IF NOT _DispatchValid() THEN
	RETURN;
ELSE
	_BuildCommandStringNoArgs();
	
	IF iBufferSend <> 0 AND __QUERYINTERFACE(iBufferSend, testIBufferSend) THEN
		iBufferSend.AddObject(RefObject := ZaberCommand);
	END_IF
END_IF
END_METHOD

METHOD set_user_vdata_3
IF ZaberStatus.ComponentStatus.iLastCommand <> 0 THEN
	ZaberStatus.ComponentStatus.iLastCommand.P_CommandStatus.LastCommandMessage := Base.F_GetLastWordInString(__POUNAME());
END_IF

IF NOT _DispatchValid() THEN
	RETURN;
ELSE
	_BuildCommandStringNoArgs();
	
	IF iBufferSend <> 0 AND __QUERYINTERFACE(iBufferSend, testIBufferSend) THEN
		iBufferSend.AddObject(RefObject := ZaberCommand);
	END_IF
END_IF
END_METHOD

METHOD set_vel
IF ZaberStatus.ComponentStatus.iLastCommand <> 0 THEN
	ZaberStatus.ComponentStatus.iLastCommand.P_CommandStatus.LastCommandMessage := Base.F_GetLastWordInString(__POUNAME());
END_IF

IF NOT _DispatchValid() THEN
	RETURN;
ELSE
	_BuildCommandStringNoArgs();
	
	IF iBufferSend <> 0 AND __QUERYINTERFACE(iBufferSend, testIBufferSend) THEN
		iBufferSend.AddObject(RefObject := ZaberCommand);
	END_IF
END_IF
END_METHOD

METHOD set_version
IF ZaberStatus.ComponentStatus.iLastCommand <> 0 THEN
	ZaberStatus.ComponentStatus.iLastCommand.P_CommandStatus.LastCommandMessage := Base.F_GetLastWordInString(__POUNAME());
END_IF

IF NOT _DispatchValid() THEN
	RETURN;
ELSE
	_BuildCommandStringNoArgs();
	
	IF iBufferSend <> 0 AND __QUERYINTERFACE(iBufferSend, testIBufferSend) THEN
		iBufferSend.AddObject(RefObject := ZaberCommand);
	END_IF
END_IF
END_METHOD

METHOD set_version_build
IF ZaberStatus.ComponentStatus.iLastCommand <> 0 THEN
	ZaberStatus.ComponentStatus.iLastCommand.P_CommandStatus.LastCommandMessage := Base.F_GetLastWordInString(__POUNAME());
END_IF

IF NOT _DispatchValid() THEN
	RETURN;
ELSE
	_BuildCommandStringNoArgs();
	
	IF iBufferSend <> 0 AND __QUERYINTERFACE(iBufferSend, testIBufferSend) THEN
		iBufferSend.AddObject(RefObject := ZaberCommand);
	END_IF
END_IF
END_METHOD

METHOD storage_append
IF ZaberStatus.ComponentStatus.iLastCommand <> 0 THEN
	ZaberStatus.ComponentStatus.iLastCommand.P_CommandStatus.LastCommandMessage := Base.F_GetLastWordInString(__POUNAME());
END_IF

IF NOT _DispatchValid() THEN
	RETURN;
ELSE
	_BuildCommandStringNoArgs();
	
	IF iBufferSend <> 0 AND __QUERYINTERFACE(iBufferSend, testIBufferSend) THEN
		iBufferSend.AddObject(RefObject := ZaberCommand);
	END_IF
END_IF
END_METHOD

METHOD storage_exists
IF ZaberStatus.ComponentStatus.iLastCommand <> 0 THEN
	ZaberStatus.ComponentStatus.iLastCommand.P_CommandStatus.LastCommandMessage := Base.F_GetLastWordInString(__POUNAME());
END_IF

IF NOT _DispatchValid() THEN
	RETURN;
ELSE
	_BuildCommandStringNoArgs();
	
	IF iBufferSend <> 0 AND __QUERYINTERFACE(iBufferSend, testIBufferSend) THEN
		iBufferSend.AddObject(RefObject := ZaberCommand);
	END_IF
END_IF
END_METHOD

METHOD storage_get
IF ZaberStatus.ComponentStatus.iLastCommand <> 0 THEN
	ZaberStatus.ComponentStatus.iLastCommand.P_CommandStatus.LastCommandMessage := Base.F_GetLastWordInString(__POUNAME());
END_IF

IF NOT _DispatchValid() THEN
	RETURN;
ELSE
	_BuildCommandStringNoArgs();
	
	IF iBufferSend <> 0 AND __QUERYINTERFACE(iBufferSend, testIBufferSend) THEN
		iBufferSend.AddObject(RefObject := ZaberCommand);
	END_IF
END_IF
END_METHOD

METHOD storage_set
IF ZaberStatus.ComponentStatus.iLastCommand <> 0 THEN
	ZaberStatus.ComponentStatus.iLastCommand.P_CommandStatus.LastCommandMessage := Base.F_GetLastWordInString(__POUNAME());
END_IF

IF NOT _DispatchValid() THEN
	RETURN;
ELSE
	_BuildCommandStringNoArgs();
	
	IF iBufferSend <> 0 AND __QUERYINTERFACE(iBufferSend, testIBufferSend) THEN
		iBufferSend.AddObject(RefObject := ZaberCommand);
	END_IF
END_IF
END_METHOD

//stream <number> [on <axis1> <axis2>] arc abs|rel cw|ccw <centrex> <centrey> <endx> <endy> [join maxspeed <speed>]; Creates an arc path segment
METHOD stream_arc
VAR_INPUT
	StreamIndex : UDINT; //<number> The number OF the stream TO ADD the ACTION TO.  Must be in the range 1 TO stream.numstreams
	Axis1 : UINT; //<axis1> The first stream axis on which TO execute the arc segment (optional).  The first stream axis is labelled "a", the second "b", AND so on
	Axis2 : UINT; //<axis2> The second stream axis on which to execute the arc segment (optional). The first stream axis is labelled "a", the second "b", and so on
	MoveType : E_MoveType; //abs Indicates that position parameters are absolute positions; rel Indicates that position parameters are relative to the end point of the previous path segment
	Direction : E_MoveDirection; //cw Indicates that the arc should be in the clockwise direction; //ccw Indicates that the arc should be in the counter-clockwise direction
	CenterX : DINT; //<centrex> The x-axis position of the arc�s centre; Must be the range -2,147,483,648 to 2,147,483,647
	CenterY : DINT; //<centrey> The y-axis position of the arc�s centre; Must be the range -2,147,483,648 to 2,147,483,647
	EndX : DINT; //<endx> The x-axis position of the end of the arc; Must be in the range limit.min to limit.max for that axis
	EndY : DINT; //<endy> The y-axis position of the end of the arc; Must be in the range limit.min to limit.max for that axis
	Speed : UDINT; //<speed> The speed LIMIT FOR the transition between the previous segment AND THIS one (optional); Must be in the range 0 TO resolution � 16,384 FOR stepper motor products; Must be in the range 0 TO 4,294,967,295 FOR linear motor OR voice coil products
END_VAR
IF ZaberStatus.ComponentStatus.iLastCommand <> 0 THEN
	ZaberStatus.ComponentStatus.iLastCommand.P_CommandStatus.LastCommandMessage := Base.F_GetLastWordInString(__POUNAME());
END_IF

IF NOT _DispatchValid() THEN
	RETURN;
ELSE
	_BuildCommandStringNoArgs();
	
	IF iBufferSend <> 0 AND __QUERYINTERFACE(iBufferSend, testIBufferSend) THEN
		iBufferSend.AddObject(RefObject := ZaberCommand);
	END_IF
END_IF
END_METHOD

METHOD stream_buffer_erase
IF ZaberStatus.ComponentStatus.iLastCommand <> 0 THEN
	ZaberStatus.ComponentStatus.iLastCommand.P_CommandStatus.LastCommandMessage := Base.F_GetLastWordInString(__POUNAME());
END_IF

IF NOT _DispatchValid() THEN
	RETURN;
ELSE
	_BuildCommandStringNoArgs();
	
	IF iBufferSend <> 0 AND __QUERYINTERFACE(iBufferSend, testIBufferSend) THEN
		iBufferSend.AddObject(RefObject := ZaberCommand);
	END_IF
END_IF
END_METHOD

METHOD stream_buffer_print
IF ZaberStatus.ComponentStatus.iLastCommand <> 0 THEN
	ZaberStatus.ComponentStatus.iLastCommand.P_CommandStatus.LastCommandMessage := Base.F_GetLastWordInString(__POUNAME());
END_IF

IF NOT _DispatchValid() THEN
	RETURN;
ELSE
	_BuildCommandStringNoArgs();
	
	IF iBufferSend <> 0 AND __QUERYINTERFACE(iBufferSend, testIBufferSend) THEN
		iBufferSend.AddObject(RefObject := ZaberCommand);
	END_IF
END_IF
END_METHOD

METHOD stream_call
IF ZaberStatus.ComponentStatus.iLastCommand <> 0 THEN
	ZaberStatus.ComponentStatus.iLastCommand.P_CommandStatus.LastCommandMessage := Base.F_GetLastWordInString(__POUNAME());
END_IF

IF NOT _DispatchValid() THEN
	RETURN;
ELSE
	_BuildCommandStringNoArgs();
	
	IF iBufferSend <> 0 AND __QUERYINTERFACE(iBufferSend, testIBufferSend) THEN
		iBufferSend.AddObject(RefObject := ZaberCommand);
	END_IF
END_IF
END_METHOD

METHOD stream_circle
IF ZaberStatus.ComponentStatus.iLastCommand <> 0 THEN
	ZaberStatus.ComponentStatus.iLastCommand.P_CommandStatus.LastCommandMessage := Base.F_GetLastWordInString(__POUNAME());
END_IF

IF NOT _DispatchValid() THEN
	RETURN;
ELSE
	_BuildCommandStringNoArgs();
	
	IF iBufferSend <> 0 AND __QUERYINTERFACE(iBufferSend, testIBufferSend) THEN
		iBufferSend.AddObject(RefObject := ZaberCommand);
	END_IF
END_IF
END_METHOD

METHOD stream_fifo
IF ZaberStatus.ComponentStatus.iLastCommand <> 0 THEN
	ZaberStatus.ComponentStatus.iLastCommand.P_CommandStatus.LastCommandMessage := Base.F_GetLastWordInString(__POUNAME());
END_IF

IF NOT _DispatchValid() THEN
	RETURN;
ELSE
	_BuildCommandStringNoArgs();
	
	IF iBufferSend <> 0 AND __QUERYINTERFACE(iBufferSend, testIBufferSend) THEN
		iBufferSend.AddObject(RefObject := ZaberCommand);
	END_IF
END_IF
END_METHOD

METHOD stream_helix
IF ZaberStatus.ComponentStatus.iLastCommand <> 0 THEN
	ZaberStatus.ComponentStatus.iLastCommand.P_CommandStatus.LastCommandMessage := Base.F_GetLastWordInString(__POUNAME());
END_IF

IF NOT _DispatchValid() THEN
	RETURN;
ELSE
	_BuildCommandStringNoArgs();
	
	IF iBufferSend <> 0 AND __QUERYINTERFACE(iBufferSend, testIBufferSend) THEN
		iBufferSend.AddObject(RefObject := ZaberCommand);
	END_IF
END_IF
END_METHOD

METHOD stream_hold_onloff
IF ZaberStatus.ComponentStatus.iLastCommand <> 0 THEN
	ZaberStatus.ComponentStatus.iLastCommand.P_CommandStatus.LastCommandMessage := Base.F_GetLastWordInString(__POUNAME());
END_IF

IF NOT _DispatchValid() THEN
	RETURN;
ELSE
	_BuildCommandStringNoArgs();
	
	IF iBufferSend <> 0 AND __QUERYINTERFACE(iBufferSend, testIBufferSend) THEN
		iBufferSend.AddObject(RefObject := ZaberCommand);
	END_IF
END_IF
END_METHOD

METHOD stream_info
IF ZaberStatus.ComponentStatus.iLastCommand <> 0 THEN
	ZaberStatus.ComponentStatus.iLastCommand.P_CommandStatus.LastCommandMessage := Base.F_GetLastWordInString(__POUNAME());
END_IF

IF NOT _DispatchValid() THEN
	RETURN;
ELSE
	_BuildCommandStringNoArgs();
	
	IF iBufferSend <> 0 AND __QUERYINTERFACE(iBufferSend, testIBufferSend) THEN
		iBufferSend.AddObject(RefObject := ZaberCommand);
	END_IF
END_IF
END_METHOD

METHOD stream_io_cancel_schedule
IF ZaberStatus.ComponentStatus.iLastCommand <> 0 THEN
	ZaberStatus.ComponentStatus.iLastCommand.P_CommandStatus.LastCommandMessage := Base.F_GetLastWordInString(__POUNAME());
END_IF

IF NOT _DispatchValid() THEN
	RETURN;
ELSE
	_BuildCommandStringNoArgs();
	
	IF iBufferSend <> 0 AND __QUERYINTERFACE(iBufferSend, testIBufferSend) THEN
		iBufferSend.AddObject(RefObject := ZaberCommand);
	END_IF
END_IF
END_METHOD

METHOD stream_io_set_ao
IF ZaberStatus.ComponentStatus.iLastCommand <> 0 THEN
	ZaberStatus.ComponentStatus.iLastCommand.P_CommandStatus.LastCommandMessage := Base.F_GetLastWordInString(__POUNAME());
END_IF

IF NOT _DispatchValid() THEN
	RETURN;
ELSE
	_BuildCommandStringNoArgs();
	
	IF iBufferSend <> 0 AND __QUERYINTERFACE(iBufferSend, testIBufferSend) THEN
		iBufferSend.AddObject(RefObject := ZaberCommand);
	END_IF
END_IF
END_METHOD

METHOD stream_io_set_ao_schedule
IF ZaberStatus.ComponentStatus.iLastCommand <> 0 THEN
	ZaberStatus.ComponentStatus.iLastCommand.P_CommandStatus.LastCommandMessage := Base.F_GetLastWordInString(__POUNAME());
END_IF

IF NOT _DispatchValid() THEN
	RETURN;
ELSE
	_BuildCommandStringNoArgs();
	
	IF iBufferSend <> 0 AND __QUERYINTERFACE(iBufferSend, testIBufferSend) THEN
		iBufferSend.AddObject(RefObject := ZaberCommand);
	END_IF
END_IF
END_METHOD

METHOD stream_io_set_do
IF ZaberStatus.ComponentStatus.iLastCommand <> 0 THEN
	ZaberStatus.ComponentStatus.iLastCommand.P_CommandStatus.LastCommandMessage := Base.F_GetLastWordInString(__POUNAME());
END_IF

IF NOT _DispatchValid() THEN
	RETURN;
ELSE
	_BuildCommandStringNoArgs();
	
	IF iBufferSend <> 0 AND __QUERYINTERFACE(iBufferSend, testIBufferSend) THEN
		iBufferSend.AddObject(RefObject := ZaberCommand);
	END_IF
END_IF
END_METHOD

METHOD stream_io_set_do_schedule
IF ZaberStatus.ComponentStatus.iLastCommand <> 0 THEN
	ZaberStatus.ComponentStatus.iLastCommand.P_CommandStatus.LastCommandMessage := Base.F_GetLastWordInString(__POUNAME());
END_IF

IF NOT _DispatchValid() THEN
	RETURN;
ELSE
	_BuildCommandStringNoArgs();
	
	IF iBufferSend <> 0 AND __QUERYINTERFACE(iBufferSend, testIBufferSend) THEN
		iBufferSend.AddObject(RefObject := ZaberCommand);
	END_IF
END_IF
END_METHOD

METHOD stream_line
IF ZaberStatus.ComponentStatus.iLastCommand <> 0 THEN
	ZaberStatus.ComponentStatus.iLastCommand.P_CommandStatus.LastCommandMessage := Base.F_GetLastWordInString(__POUNAME());
END_IF

IF NOT _DispatchValid() THEN
	RETURN;
ELSE
	_BuildCommandStringNoArgs();
	
	IF iBufferSend <> 0 AND __QUERYINTERFACE(iBufferSend, testIBufferSend) THEN
		iBufferSend.AddObject(RefObject := ZaberCommand);
	END_IF
END_IF
END_METHOD

METHOD stream_set
IF ZaberStatus.ComponentStatus.iLastCommand <> 0 THEN
	ZaberStatus.ComponentStatus.iLastCommand.P_CommandStatus.LastCommandMessage := Base.F_GetLastWordInString(__POUNAME());
END_IF

IF NOT _DispatchValid() THEN
	RETURN;
ELSE
	_BuildCommandStringNoArgs();
	
	IF iBufferSend <> 0 AND __QUERYINTERFACE(iBufferSend, testIBufferSend) THEN
		iBufferSend.AddObject(RefObject := ZaberCommand);
	END_IF
END_IF
END_METHOD

METHOD stream_setup_disable
IF ZaberStatus.ComponentStatus.iLastCommand <> 0 THEN
	ZaberStatus.ComponentStatus.iLastCommand.P_CommandStatus.LastCommandMessage := Base.F_GetLastWordInString(__POUNAME());
END_IF

IF NOT _DispatchValid() THEN
	RETURN;
ELSE
	_BuildCommandStringNoArgs();
	
	IF iBufferSend <> 0 AND __QUERYINTERFACE(iBufferSend, testIBufferSend) THEN
		iBufferSend.AddObject(RefObject := ZaberCommand);
	END_IF
END_IF
END_METHOD

METHOD stream_setup_live
VAR_INPUT
	StreamNumber : UDINT;
	AxisNumber : UDINT;
END_VAR
IF ZaberStatus.ComponentStatus.iLastCommand <> 0 THEN
	ZaberStatus.ComponentStatus.iLastCommand.P_CommandStatus.LastCommandMessage := Base.F_GetLastWordInString(__POUNAME());
END_IF

IF NOT _DispatchValid() THEN
	RETURN;
ELSE
	_ClearTempString();
	ZaberCommand.stringval := Tc2_Standard.CONCAT(STR1 := ZaberConfiguration.sControllerRef, STR2 := ' ');
	ZaberCommand.stringval := Tc2_Standard.CONCAT(STR1 := ZaberCommand.stringval, STR2 := UINT_TO_STRING(ZaberConfiguration.AxisRef));
	ZaberCommand.stringval := Tc2_Standard.CONCAT(STR1 := ZaberCommand.stringval, STR2 := ' ');
	ZaberCommand.stringval := Tc2_Standard.CONCAT(STR1 := ZaberCommand.stringval, STR2 := Base.F_GetFirstWordInString(SUPER^._iCommandConfiguration[ZaberStatus.ZaberMethodDispatch].P_CommandConfiguration.CommandDescription));
	ZaberCommand.stringval := Tc2_Standard.CONCAT(STR1 := ZaberCommand.stringval, STR2 := ' ');
	ZaberCommand.stringval := Tc2_Standard.CONCAT(STR1 := ZaberCommand.stringval, STR2 := UDINT_TO_STRING(StreamNumber));
	ZaberCommand.stringval := Tc2_Standard.CONCAT(STR1 := ZaberCommand.stringval, STR2 := ' ');
	ZaberCommand.stringval := Tc2_Standard.CONCAT(STR1 := ZaberCommand.stringval, STR2 := F_GetAllButFirstWord(SUPER^._iCommandConfiguration[ZaberStatus.ZaberMethodDispatch].P_CommandConfiguration.CommandDescription));
	ZaberCommand.stringval := Tc2_Standard.CONCAT(STR1 := ZaberCommand.stringval, STR2 := ' ');
	ZaberCommand.stringval := Tc2_Standard.CONCAT(STR1 := ZaberCommand.stringval, STR2 := UDINT_TO_STRING(AxisNumber));

	IF iBufferSend <> 0 AND __QUERYINTERFACE(iBufferSend, testIBufferSend) THEN
		iBufferSend.AddObject(RefObject := ZaberCommand);
	END_IF
END_IF
END_METHOD

METHOD stream_setup_store
VAR_INPUT
	StreamNumber	: UDINT; //The number OF the stream TO enable; Must be in the range 1 TO stream.numstreams
	BufferNumber	: UDINT; //The number OF the buffer TO write TO; Must be in the range 1 to stream.numbufs
	AxisNumber		: UINT; //The number OF axes in the path ; Must be in the range 1 TO system.axiscount
END_VAR
IF ZaberStatus.ComponentStatus.iLastCommand <> 0 THEN
	ZaberStatus.ComponentStatus.iLastCommand.P_CommandStatus.LastCommandMessage := Base.F_GetLastWordInString(__POUNAME());
END_IF

IF NOT _DispatchValid() THEN
	RETURN;
ELSE
	_ClearTempString();
	ZaberCommand.stringval := Tc2_Standard.CONCAT(STR1 := ZaberConfiguration.sControllerRef, STR2 := ' ');
	ZaberCommand.stringval := Tc2_Standard.CONCAT(STR1 := ZaberCommand.stringval, STR2 := UINT_TO_STRING(ZaberConfiguration.AxisRef));
	ZaberCommand.stringval := Tc2_Standard.CONCAT(STR1 := ZaberCommand.stringval, STR2 := ' ');
	ZaberCommand.stringval := Tc2_Standard.CONCAT(STR1 := ZaberCommand.stringval, STR2 := Base.F_GetFirstWordInString(SUPER^._iCommandConfiguration[ZaberStatus.ZaberMethodDispatch].P_CommandConfiguration.CommandDescription));
	ZaberCommand.stringval := Tc2_Standard.CONCAT(STR1 := ZaberCommand.stringval, STR2 := ' ');
	ZaberCommand.stringval := Tc2_Standard.CONCAT(STR1 := ZaberCommand.stringval, STR2 := UDINT_TO_STRING(StreamNumber));
	ZaberCommand.stringval := Tc2_Standard.CONCAT(STR1 := ZaberCommand.stringval, STR2 := ' ');
	ZaberCommand.stringval := Tc2_Standard.CONCAT(STR1 := ZaberCommand.stringval, STR2 := F_GetAllButFirstWord(SUPER^._iCommandConfiguration[ZaberStatus.ZaberMethodDispatch].P_CommandConfiguration.CommandDescription));
	ZaberCommand.stringval := Tc2_Standard.CONCAT(STR1 := ZaberCommand.stringval, STR2 := ' ');
	ZaberCommand.stringval := Tc2_Standard.CONCAT(STR1 := ZaberCommand.stringval, STR2 := UDINT_TO_STRING(BufferNumber));
	ZaberCommand.stringval := Tc2_Standard.CONCAT(STR1 := ZaberCommand.stringval, STR2 := ' ');
	ZaberCommand.stringval := Tc2_Standard.CONCAT(STR1 := ZaberCommand.stringval, STR2 := UINT_TO_STRING(AxisNumber));
	
	IF iBufferSend <> 0 AND __QUERYINTERFACE(iBufferSend, testIBufferSend) THEN
		iBufferSend.AddObject(RefObject := ZaberCommand);
	END_IF
END_IF
END_METHOD

METHOD stream_wait
IF ZaberStatus.ComponentStatus.iLastCommand <> 0 THEN
	ZaberStatus.ComponentStatus.iLastCommand.P_CommandStatus.LastCommandMessage := Base.F_GetLastWordInString(__POUNAME());
END_IF

IF NOT _DispatchValid() THEN
	RETURN;
ELSE
	_BuildCommandStringNoArgs();
	
	IF iBufferSend <> 0 AND __QUERYINTERFACE(iBufferSend, testIBufferSend) THEN
		iBufferSend.AddObject(RefObject := ZaberCommand);
	END_IF
END_IF
END_METHOD

METHOD stream_wait_io
IF ZaberStatus.ComponentStatus.iLastCommand <> 0 THEN
	ZaberStatus.ComponentStatus.iLastCommand.P_CommandStatus.LastCommandMessage := Base.F_GetLastWordInString(__POUNAME());
END_IF

IF NOT _DispatchValid() THEN
	RETURN;
ELSE
	_BuildCommandStringNoArgs();
	
	IF iBufferSend <> 0 AND __QUERYINTERFACE(iBufferSend, testIBufferSend) THEN
		iBufferSend.AddObject(RefObject := ZaberCommand);
	END_IF
END_IF
END_METHOD

METHOD tools_storepos
IF ZaberStatus.ComponentStatus.iLastCommand <> 0 THEN
	ZaberStatus.ComponentStatus.iLastCommand.P_CommandStatus.LastCommandMessage := Base.F_GetLastWordInString(__POUNAME());
END_IF

IF NOT _DispatchValid() THEN
	RETURN;
ELSE
	_BuildCommandStringNoArgs();
	
	IF iBufferSend <> 0 AND __QUERYINTERFACE(iBufferSend, testIBufferSend) THEN
		iBufferSend.AddObject(RefObject := ZaberCommand);
	END_IF
END_IF
END_METHOD

METHOD trigger_action_command
IF ZaberStatus.ComponentStatus.iLastCommand <> 0 THEN
	ZaberStatus.ComponentStatus.iLastCommand.P_CommandStatus.LastCommandMessage := Base.F_GetLastWordInString(__POUNAME());
END_IF

IF NOT _DispatchValid() THEN
	RETURN;
ELSE
	_BuildCommandStringNoArgs();
	
	IF iBufferSend <> 0 AND __QUERYINTERFACE(iBufferSend, testIBufferSend) THEN
		iBufferSend.AddObject(RefObject := ZaberCommand);
	END_IF
END_IF
END_METHOD

METHOD trigger_action_none
IF ZaberStatus.ComponentStatus.iLastCommand <> 0 THEN
	ZaberStatus.ComponentStatus.iLastCommand.P_CommandStatus.LastCommandMessage := Base.F_GetLastWordInString(__POUNAME());
END_IF

IF NOT _DispatchValid() THEN
	RETURN;
ELSE
	_BuildCommandStringNoArgs();
	
	IF iBufferSend <> 0 AND __QUERYINTERFACE(iBufferSend, testIBufferSend) THEN
		iBufferSend.AddObject(RefObject := ZaberCommand);
	END_IF
END_IF
END_METHOD

METHOD trigger_action_setting
IF ZaberStatus.ComponentStatus.iLastCommand <> 0 THEN
	ZaberStatus.ComponentStatus.iLastCommand.P_CommandStatus.LastCommandMessage := Base.F_GetLastWordInString(__POUNAME());
END_IF

IF NOT _DispatchValid() THEN
	RETURN;
ELSE
	_BuildCommandStringNoArgs();
	
	IF iBufferSend <> 0 AND __QUERYINTERFACE(iBufferSend, testIBufferSend) THEN
		iBufferSend.AddObject(RefObject := ZaberCommand);
	END_IF
END_IF
END_METHOD

METHOD trigger_disable
IF ZaberStatus.ComponentStatus.iLastCommand <> 0 THEN
	ZaberStatus.ComponentStatus.iLastCommand.P_CommandStatus.LastCommandMessage := Base.F_GetLastWordInString(__POUNAME());
END_IF

IF NOT _DispatchValid() THEN
	RETURN;
ELSE
	_BuildCommandStringNoArgs();
	
	IF iBufferSend <> 0 AND __QUERYINTERFACE(iBufferSend, testIBufferSend) THEN
		iBufferSend.AddObject(RefObject := ZaberCommand);
	END_IF
END_IF
END_METHOD

METHOD trigger_enable
IF ZaberStatus.ComponentStatus.iLastCommand <> 0 THEN
	ZaberStatus.ComponentStatus.iLastCommand.P_CommandStatus.LastCommandMessage := Base.F_GetLastWordInString(__POUNAME());
END_IF

IF NOT _DispatchValid() THEN
	RETURN;
ELSE
	_BuildCommandStringNoArgs();
	
	IF iBufferSend <> 0 AND __QUERYINTERFACE(iBufferSend, testIBufferSend) THEN
		iBufferSend.AddObject(RefObject := ZaberCommand);
	END_IF
END_IF
END_METHOD

METHOD trigger_when_io
IF ZaberStatus.ComponentStatus.iLastCommand <> 0 THEN
	ZaberStatus.ComponentStatus.iLastCommand.P_CommandStatus.LastCommandMessage := Base.F_GetLastWordInString(__POUNAME());
END_IF

IF NOT _DispatchValid() THEN
	RETURN;
ELSE
	_BuildCommandStringNoArgs();
	
	IF iBufferSend <> 0 AND __QUERYINTERFACE(iBufferSend, testIBufferSend) THEN
		iBufferSend.AddObject(RefObject := ZaberCommand);
	END_IF
END_IF
END_METHOD

METHOD trigger_when_setting
IF ZaberStatus.ComponentStatus.iLastCommand <> 0 THEN
	ZaberStatus.ComponentStatus.iLastCommand.P_CommandStatus.LastCommandMessage := Base.F_GetLastWordInString(__POUNAME());
END_IF

IF NOT _DispatchValid() THEN
	RETURN;
ELSE
	_BuildCommandStringNoArgs();
	
	IF iBufferSend <> 0 AND __QUERYINTERFACE(iBufferSend, testIBufferSend) THEN
		iBufferSend.AddObject(RefObject := ZaberCommand);
	END_IF
END_IF
END_METHOD

METHOD trigger_when_time
IF ZaberStatus.ComponentStatus.iLastCommand <> 0 THEN
	ZaberStatus.ComponentStatus.iLastCommand.P_CommandStatus.LastCommandMessage := Base.F_GetLastWordInString(__POUNAME());
END_IF

IF NOT _DispatchValid() THEN
	RETURN;
ELSE
	_BuildCommandStringNoArgs();
	
	IF iBufferSend <> 0 AND __QUERYINTERFACE(iBufferSend, testIBufferSend) THEN
		iBufferSend.AddObject(RefObject := ZaberCommand);
	END_IF
END_IF
END_METHOD

METHOD activate
IF ZaberStatus.ComponentStatus.iLastCommand <> 0 THEN
	ZaberStatus.ComponentStatus.iLastCommand.P_CommandStatus.LastCommandMessage := Base.F_GetLastWordInString(__POUNAME());
END_IF

IF NOT _DispatchValid() THEN
	RETURN;
ELSE
	_BuildCommandStringNoArgs();
	
	IF iBufferSend <> 0 AND __QUERYINTERFACE(iBufferSend, testIBufferSend) THEN
		iBufferSend.AddObject(RefObject := ZaberCommand);
	END_IF
END_IF
END_METHOD

METHOD axis_restore
IF ZaberStatus.ComponentStatus.iLastCommand <> 0 THEN
	ZaberStatus.ComponentStatus.iLastCommand.P_CommandStatus.LastCommandMessage := Base.F_GetLastWordInString(__POUNAME());
END_IF

IF NOT _DispatchValid() THEN
	RETURN;
ELSE
	_BuildCommandStringNoArgs();
	
	IF iBufferSend <> 0 AND __QUERYINTERFACE(iBufferSend, testIBufferSend) THEN
		iBufferSend.AddObject(RefObject := ZaberCommand);
	END_IF
END_IF
END_METHOD

METHOD comm_en_ipv4_dhcp
IF ZaberStatus.ComponentStatus.iLastCommand <> 0 THEN
	ZaberStatus.ComponentStatus.iLastCommand.P_CommandStatus.LastCommandMessage := Base.F_GetLastWordInString(__POUNAME());
END_IF

IF NOT _DispatchValid() THEN
	RETURN;
ELSE
	_BuildCommandStringNoArgs();
	
	IF iBufferSend <> 0 AND __QUERYINTERFACE(iBufferSend, testIBufferSend) THEN
		iBufferSend.AddObject(RefObject := ZaberCommand);
	END_IF
END_IF
END_METHOD

METHOD driver_disable
IF ZaberStatus.ComponentStatus.iLastCommand <> 0 THEN
	ZaberStatus.ComponentStatus.iLastCommand.P_CommandStatus.LastCommandMessage := Base.F_GetLastWordInString(__POUNAME());
END_IF

IF NOT _DispatchValid() THEN
	RETURN;
ELSE
	_BuildCommandStringNoArgs();
	
	IF iBufferSend <> 0 AND __QUERYINTERFACE(iBufferSend, testIBufferSend) THEN
		iBufferSend.AddObject(RefObject := ZaberCommand);
	END_IF
END_IF
END_METHOD

METHOD driver_enable
IF ZaberStatus.ComponentStatus.iLastCommand <> 0 THEN
	ZaberStatus.ComponentStatus.iLastCommand.P_CommandStatus.LastCommandMessage := Base.F_GetLastWordInString(__POUNAME());
END_IF

IF NOT _DispatchValid() THEN
	RETURN;
ELSE
	_BuildCommandStringNoArgs();
	
	IF iBufferSend <> 0 AND __QUERYINTERFACE(iBufferSend, testIBufferSend) THEN
		iBufferSend.AddObject(RefObject := ZaberCommand);
	END_IF
END_IF
END_METHOD

METHOD get_accel
IF ZaberStatus.ComponentStatus.iLastCommand <> 0 THEN
	ZaberStatus.ComponentStatus.iLastCommand.P_CommandStatus.LastCommandMessage := Base.F_GetLastWordInString(__POUNAME());
END_IF

IF NOT _DispatchValid() THEN
	RETURN;
ELSE
	_BuildCommandStringNoArgs();
	
	IF iBufferSend <> 0 AND __QUERYINTERFACE(iBufferSend, testIBufferSend) THEN
		iBufferSend.AddObject(RefObject := ZaberCommand);
	END_IF
END_IF
END_METHOD

METHOD get_autodetect_coil_mode
IF ZaberStatus.ComponentStatus.iLastCommand <> 0 THEN
	ZaberStatus.ComponentStatus.iLastCommand.P_CommandStatus.LastCommandMessage := Base.F_GetLastWordInString(__POUNAME());
END_IF

IF NOT _DispatchValid() THEN
	RETURN;
ELSE
	_BuildCommandStringNoArgs();
	
	IF iBufferSend <> 0 AND __QUERYINTERFACE(iBufferSend, testIBufferSend) THEN
		iBufferSend.AddObject(RefObject := ZaberCommand);
	END_IF
END_IF
END_METHOD

METHOD get_calibration_type
IF ZaberStatus.ComponentStatus.iLastCommand <> 0 THEN
	ZaberStatus.ComponentStatus.iLastCommand.P_CommandStatus.LastCommandMessage := Base.F_GetLastWordInString(__POUNAME());
END_IF

IF NOT _DispatchValid() THEN
	RETURN;
ELSE
	_BuildCommandStringNoArgs();
	
	IF iBufferSend <> 0 AND __QUERYINTERFACE(iBufferSend, testIBufferSend) THEN
		iBufferSend.AddObject(RefObject := ZaberCommand);
	END_IF
END_IF
END_METHOD

METHOD get_comm_address
IF ZaberStatus.ComponentStatus.iLastCommand <> 0 THEN
	ZaberStatus.ComponentStatus.iLastCommand.P_CommandStatus.LastCommandMessage := Base.F_GetLastWordInString(__POUNAME());
END_IF

IF NOT _DispatchValid() THEN
	RETURN;
ELSE
	_BuildCommandStringNoArgs();
	
	IF iBufferSend <> 0 AND __QUERYINTERFACE(iBufferSend, testIBufferSend) THEN
		iBufferSend.AddObject(RefObject := ZaberCommand);
	END_IF
END_IF
END_METHOD

METHOD get_comm_alert
IF ZaberStatus.ComponentStatus.iLastCommand <> 0 THEN
	ZaberStatus.ComponentStatus.iLastCommand.P_CommandStatus.LastCommandMessage := Base.F_GetLastWordInString(__POUNAME());
END_IF

IF NOT _DispatchValid() THEN
	RETURN;
ELSE
	_BuildCommandStringNoArgs();
	
	IF iBufferSend <> 0 AND __QUERYINTERFACE(iBufferSend, testIBufferSend) THEN
		iBufferSend.AddObject(RefObject := ZaberCommand);
	END_IF
END_IF
END_METHOD

METHOD get_comm_checksum
IF ZaberStatus.ComponentStatus.iLastCommand <> 0 THEN
	ZaberStatus.ComponentStatus.iLastCommand.P_CommandStatus.LastCommandMessage := Base.F_GetLastWordInString(__POUNAME());
END_IF

IF NOT _DispatchValid() THEN
	RETURN;
ELSE
	_BuildCommandStringNoArgs();
	
	IF iBufferSend <> 0 AND __QUERYINTERFACE(iBufferSend, testIBufferSend) THEN
		iBufferSend.AddObject(RefObject := ZaberCommand);
	END_IF
END_IF
END_METHOD

METHOD get_comm_command_packets_max
IF ZaberStatus.ComponentStatus.iLastCommand <> 0 THEN
	ZaberStatus.ComponentStatus.iLastCommand.P_CommandStatus.LastCommandMessage := Base.F_GetLastWordInString(__POUNAME());
END_IF

IF NOT _DispatchValid() THEN
	RETURN;
ELSE
	_BuildCommandStringNoArgs();
	
	IF iBufferSend <> 0 AND __QUERYINTERFACE(iBufferSend, testIBufferSend) THEN
		iBufferSend.AddObject(RefObject := ZaberCommand);
	END_IF
END_IF
END_METHOD

METHOD get_comm_en_ipv4_address
IF ZaberStatus.ComponentStatus.iLastCommand <> 0 THEN
	ZaberStatus.ComponentStatus.iLastCommand.P_CommandStatus.LastCommandMessage := Base.F_GetLastWordInString(__POUNAME());
END_IF

IF NOT _DispatchValid() THEN
	RETURN;
ELSE
	_BuildCommandStringNoArgs();
	
	IF iBufferSend <> 0 AND __QUERYINTERFACE(iBufferSend, testIBufferSend) THEN
		iBufferSend.AddObject(RefObject := ZaberCommand);
	END_IF
END_IF
END_METHOD

METHOD get_comm_en_ipv4_dhcp_enabled
IF ZaberStatus.ComponentStatus.iLastCommand <> 0 THEN
	ZaberStatus.ComponentStatus.iLastCommand.P_CommandStatus.LastCommandMessage := Base.F_GetLastWordInString(__POUNAME());
END_IF

IF NOT _DispatchValid() THEN
	RETURN;
ELSE
	_BuildCommandStringNoArgs();
	
	IF iBufferSend <> 0 AND __QUERYINTERFACE(iBufferSend, testIBufferSend) THEN
		iBufferSend.AddObject(RefObject := ZaberCommand);
	END_IF
END_IF
END_METHOD

METHOD get_comm_en_ipv4_gateway
IF ZaberStatus.ComponentStatus.iLastCommand <> 0 THEN
	ZaberStatus.ComponentStatus.iLastCommand.P_CommandStatus.LastCommandMessage := Base.F_GetLastWordInString(__POUNAME());
END_IF

IF NOT _DispatchValid() THEN
	RETURN;
ELSE
	_BuildCommandStringNoArgs();
	
	IF iBufferSend <> 0 AND __QUERYINTERFACE(iBufferSend, testIBufferSend) THEN
		iBufferSend.AddObject(RefObject := ZaberCommand);
	END_IF
END_IF
END_METHOD

METHOD get_comm_en_ipv4_netmask
IF ZaberStatus.ComponentStatus.iLastCommand <> 0 THEN
	ZaberStatus.ComponentStatus.iLastCommand.P_CommandStatus.LastCommandMessage := Base.F_GetLastWordInString(__POUNAME());
END_IF

IF NOT _DispatchValid() THEN
	RETURN;
ELSE
	_BuildCommandStringNoArgs();
	
	IF iBufferSend <> 0 AND __QUERYINTERFACE(iBufferSend, testIBufferSend) THEN
		iBufferSend.AddObject(RefObject := ZaberCommand);
	END_IF
END_IF
END_METHOD

METHOD get_comm_en_mac
IF ZaberStatus.ComponentStatus.iLastCommand <> 0 THEN
	ZaberStatus.ComponentStatus.iLastCommand.P_CommandStatus.LastCommandMessage := Base.F_GetLastWordInString(__POUNAME());
END_IF

IF NOT _DispatchValid() THEN
	RETURN;
ELSE
	_BuildCommandStringNoArgs();
	
	IF iBufferSend <> 0 AND __QUERYINTERFACE(iBufferSend, testIBufferSend) THEN
		iBufferSend.AddObject(RefObject := ZaberCommand);
	END_IF
END_IF
END_METHOD

METHOD get_comm_en_mdns_enable
IF ZaberStatus.ComponentStatus.iLastCommand <> 0 THEN
	ZaberStatus.ComponentStatus.iLastCommand.P_CommandStatus.LastCommandMessage := Base.F_GetLastWordInString(__POUNAME());
END_IF

IF NOT _DispatchValid() THEN
	RETURN;
ELSE
	_BuildCommandStringNoArgs();
	
	IF iBufferSend <> 0 AND __QUERYINTERFACE(iBufferSend, testIBufferSend) THEN
		iBufferSend.AddObject(RefObject := ZaberCommand);
	END_IF
END_IF
END_METHOD

METHOD get_comm_next_owner
IF ZaberStatus.ComponentStatus.iLastCommand <> 0 THEN
	ZaberStatus.ComponentStatus.iLastCommand.P_CommandStatus.LastCommandMessage := Base.F_GetLastWordInString(__POUNAME());
END_IF

IF NOT _DispatchValid() THEN
	RETURN;
ELSE
	_BuildCommandStringNoArgs();
	
	IF iBufferSend <> 0 AND __QUERYINTERFACE(iBufferSend, testIBufferSend) THEN
		iBufferSend.AddObject(RefObject := ZaberCommand);
	END_IF
END_IF
END_METHOD

METHOD get_comm_packet_size_max
IF ZaberStatus.ComponentStatus.iLastCommand <> 0 THEN
	ZaberStatus.ComponentStatus.iLastCommand.P_CommandStatus.LastCommandMessage := Base.F_GetLastWordInString(__POUNAME());
END_IF

IF NOT _DispatchValid() THEN
	RETURN;
ELSE
	_BuildCommandStringNoArgs();
	
	IF iBufferSend <> 0 AND __QUERYINTERFACE(iBufferSend, testIBufferSend) THEN
		iBufferSend.AddObject(RefObject := ZaberCommand);
	END_IF
END_IF
END_METHOD

METHOD get_comm_protocol
IF ZaberStatus.ComponentStatus.iLastCommand <> 0 THEN
	ZaberStatus.ComponentStatus.iLastCommand.P_CommandStatus.LastCommandMessage := Base.F_GetLastWordInString(__POUNAME());
END_IF

IF NOT _DispatchValid() THEN
	RETURN;
ELSE
	_BuildCommandStringNoArgs();
	
	IF iBufferSend <> 0 AND __QUERYINTERFACE(iBufferSend, testIBufferSend) THEN
		iBufferSend.AddObject(RefObject := ZaberCommand);
	END_IF
END_IF
END_METHOD

METHOD get_comm_rs232_baud
IF ZaberStatus.ComponentStatus.iLastCommand <> 0 THEN
	ZaberStatus.ComponentStatus.iLastCommand.P_CommandStatus.LastCommandMessage := Base.F_GetLastWordInString(__POUNAME());
END_IF

IF NOT _DispatchValid() THEN
	RETURN;
ELSE
	_BuildCommandStringNoArgs();
	
	IF iBufferSend <> 0 AND __QUERYINTERFACE(iBufferSend, testIBufferSend) THEN
		iBufferSend.AddObject(RefObject := ZaberCommand);
	END_IF
END_IF
END_METHOD

METHOD get_comm_word_size_max
IF ZaberStatus.ComponentStatus.iLastCommand <> 0 THEN
	ZaberStatus.ComponentStatus.iLastCommand.P_CommandStatus.LastCommandMessage := Base.F_GetLastWordInString(__POUNAME());
END_IF

IF NOT _DispatchValid() THEN
	RETURN;
ELSE
	_BuildCommandStringNoArgs();
	
	IF iBufferSend <> 0 AND __QUERYINTERFACE(iBufferSend, testIBufferSend) THEN
		iBufferSend.AddObject(RefObject := ZaberCommand);
	END_IF
END_IF
END_METHOD

METHOD get_device_hw_modified
IF ZaberStatus.ComponentStatus.iLastCommand <> 0 THEN
	ZaberStatus.ComponentStatus.iLastCommand.P_CommandStatus.LastCommandMessage := Base.F_GetLastWordInString(__POUNAME());
END_IF

IF NOT _DispatchValid() THEN
	RETURN;
ELSE
	_BuildCommandStringNoArgs();
	
	IF iBufferSend <> 0 AND __QUERYINTERFACE(iBufferSend, testIBufferSend) THEN
		iBufferSend.AddObject(RefObject := ZaberCommand);
	END_IF
END_IF
END_METHOD

METHOD get_device_id
IF ZaberStatus.ComponentStatus.iLastCommand <> 0 THEN
	ZaberStatus.ComponentStatus.iLastCommand.P_CommandStatus.LastCommandMessage := Base.F_GetLastWordInString(__POUNAME());
END_IF

IF NOT _DispatchValid() THEN
	RETURN;
ELSE
	_BuildCommandStringNoArgs();
	
	IF iBufferSend <> 0 AND __QUERYINTERFACE(iBufferSend, testIBufferSend) THEN
		iBufferSend.AddObject(RefObject := ZaberCommand);
	END_IF
END_IF
END_METHOD

METHOD get_driver_current_approach
IF ZaberStatus.ComponentStatus.iLastCommand <> 0 THEN
	ZaberStatus.ComponentStatus.iLastCommand.P_CommandStatus.LastCommandMessage := Base.F_GetLastWordInString(__POUNAME());
END_IF

IF NOT _DispatchValid() THEN
	RETURN;
ELSE
	_BuildCommandStringNoArgs();
	
	IF iBufferSend <> 0 AND __QUERYINTERFACE(iBufferSend, testIBufferSend) THEN
		iBufferSend.AddObject(RefObject := ZaberCommand);
	END_IF
END_IF
END_METHOD

METHOD get_driver_current_hold
IF ZaberStatus.ComponentStatus.iLastCommand <> 0 THEN
	ZaberStatus.ComponentStatus.iLastCommand.P_CommandStatus.LastCommandMessage := Base.F_GetLastWordInString(__POUNAME());
END_IF

IF NOT _DispatchValid() THEN
	RETURN;
ELSE
	_BuildCommandStringNoArgs();
	
	IF iBufferSend <> 0 AND __QUERYINTERFACE(iBufferSend, testIBufferSend) THEN
		iBufferSend.AddObject(RefObject := ZaberCommand);
	END_IF
END_IF
END_METHOD

METHOD get_driver_current_max
IF ZaberStatus.ComponentStatus.iLastCommand <> 0 THEN
	ZaberStatus.ComponentStatus.iLastCommand.P_CommandStatus.LastCommandMessage := Base.F_GetLastWordInString(__POUNAME());
END_IF

IF NOT _DispatchValid() THEN
	RETURN;
ELSE
	_BuildCommandStringNoArgs();
	
	IF iBufferSend <> 0 AND __QUERYINTERFACE(iBufferSend, testIBufferSend) THEN
		iBufferSend.AddObject(RefObject := ZaberCommand);
	END_IF
END_IF
END_METHOD

METHOD get_driver_current_run
IF ZaberStatus.ComponentStatus.iLastCommand <> 0 THEN
	ZaberStatus.ComponentStatus.iLastCommand.P_CommandStatus.LastCommandMessage := Base.F_GetLastWordInString(__POUNAME());
END_IF

IF NOT _DispatchValid() THEN
	RETURN;
ELSE
	_BuildCommandStringNoArgs();
	
	IF iBufferSend <> 0 AND __QUERYINTERFACE(iBufferSend, testIBufferSend) THEN
		iBufferSend.AddObject(RefObject := ZaberCommand);
	END_IF
END_IF
END_METHOD

METHOD get_driver_enable_mode
IF ZaberStatus.ComponentStatus.iLastCommand <> 0 THEN
	ZaberStatus.ComponentStatus.iLastCommand.P_CommandStatus.LastCommandMessage := Base.F_GetLastWordInString(__POUNAME());
END_IF

IF NOT _DispatchValid() THEN
	RETURN;
ELSE
	_BuildCommandStringNoArgs();
	
	IF iBufferSend <> 0 AND __QUERYINTERFACE(iBufferSend, testIBufferSend) THEN
		iBufferSend.AddObject(RefObject := ZaberCommand);
	END_IF
END_IF
END_METHOD

METHOD get_driver_enabled
IF ZaberStatus.ComponentStatus.iLastCommand <> 0 THEN
	ZaberStatus.ComponentStatus.iLastCommand.P_CommandStatus.LastCommandMessage := Base.F_GetLastWordInString(__POUNAME());
END_IF

IF NOT _DispatchValid() THEN
	RETURN;
ELSE
	_BuildCommandStringNoArgs();
	
	IF iBufferSend <> 0 AND __QUERYINTERFACE(iBufferSend, testIBufferSend) THEN
		iBufferSend.AddObject(RefObject := ZaberCommand);
	END_IF
END_IF
END_METHOD

METHOD get_driver_temperature
IF ZaberStatus.ComponentStatus.iLastCommand <> 0 THEN
	ZaberStatus.ComponentStatus.iLastCommand.P_CommandStatus.LastCommandMessage := Base.F_GetLastWordInString(__POUNAME());
END_IF

IF NOT _DispatchValid() THEN
	RETURN;
ELSE
	_BuildCommandStringNoArgs();
	
	IF iBufferSend <> 0 AND __QUERYINTERFACE(iBufferSend, testIBufferSend) THEN
		iBufferSend.AddObject(RefObject := ZaberCommand);
	END_IF
END_IF
END_METHOD

METHOD get_get_settings_max
IF ZaberStatus.ComponentStatus.iLastCommand <> 0 THEN
	ZaberStatus.ComponentStatus.iLastCommand.P_CommandStatus.LastCommandMessage := Base.F_GetLastWordInString(__POUNAME());
END_IF

IF NOT _DispatchValid() THEN
	RETURN;
ELSE
	_BuildCommandStringNoArgs();
	
	IF iBufferSend <> 0 AND __QUERYINTERFACE(iBufferSend, testIBufferSend) THEN
		iBufferSend.AddObject(RefObject := ZaberCommand);
	END_IF
END_IF
END_METHOD

METHOD get_ictrl_advance_a
IF ZaberStatus.ComponentStatus.iLastCommand <> 0 THEN
	ZaberStatus.ComponentStatus.iLastCommand.P_CommandStatus.LastCommandMessage := Base.F_GetLastWordInString(__POUNAME());
END_IF

IF NOT _DispatchValid() THEN
	RETURN;
ELSE
	_BuildCommandStringNoArgs();
	
	IF iBufferSend <> 0 AND __QUERYINTERFACE(iBufferSend, testIBufferSend) THEN
		iBufferSend.AddObject(RefObject := ZaberCommand);
	END_IF
END_IF
END_METHOD

METHOD get_ictrl_advance_offset
IF ZaberStatus.ComponentStatus.iLastCommand <> 0 THEN
	ZaberStatus.ComponentStatus.iLastCommand.P_CommandStatus.LastCommandMessage := Base.F_GetLastWordInString(__POUNAME());
END_IF

IF NOT _DispatchValid() THEN
	RETURN;
ELSE
	_BuildCommandStringNoArgs();
	
	IF iBufferSend <> 0 AND __QUERYINTERFACE(iBufferSend, testIBufferSend) THEN
		iBufferSend.AddObject(RefObject := ZaberCommand);
	END_IF
END_IF
END_METHOD

METHOD get_ictrl_afcff_inductance
IF ZaberStatus.ComponentStatus.iLastCommand <> 0 THEN
	ZaberStatus.ComponentStatus.iLastCommand.P_CommandStatus.LastCommandMessage := Base.F_GetLastWordInString(__POUNAME());
END_IF

IF NOT _DispatchValid() THEN
	RETURN;
ELSE
	_BuildCommandStringNoArgs();
	
	IF iBufferSend <> 0 AND __QUERYINTERFACE(iBufferSend, testIBufferSend) THEN
		iBufferSend.AddObject(RefObject := ZaberCommand);
	END_IF
END_IF
END_METHOD

METHOD get_ictrl_afcff_ke
IF ZaberStatus.ComponentStatus.iLastCommand <> 0 THEN
	ZaberStatus.ComponentStatus.iLastCommand.P_CommandStatus.LastCommandMessage := Base.F_GetLastWordInString(__POUNAME());
END_IF

IF NOT _DispatchValid() THEN
	RETURN;
ELSE
	_BuildCommandStringNoArgs();
	
	IF iBufferSend <> 0 AND __QUERYINTERFACE(iBufferSend, testIBufferSend) THEN
		iBufferSend.AddObject(RefObject := ZaberCommand);
	END_IF
END_IF
END_METHOD

METHOD get_ictrl_afcff_ki
IF ZaberStatus.ComponentStatus.iLastCommand <> 0 THEN
	ZaberStatus.ComponentStatus.iLastCommand.P_CommandStatus.LastCommandMessage := Base.F_GetLastWordInString(__POUNAME());
END_IF

IF NOT _DispatchValid() THEN
	RETURN;
ELSE
	_BuildCommandStringNoArgs();
	
	IF iBufferSend <> 0 AND __QUERYINTERFACE(iBufferSend, testIBufferSend) THEN
		iBufferSend.AddObject(RefObject := ZaberCommand);
	END_IF
END_IF
END_METHOD

METHOD get_ictrl_afcff_max
IF ZaberStatus.ComponentStatus.iLastCommand <> 0 THEN
	ZaberStatus.ComponentStatus.iLastCommand.P_CommandStatus.LastCommandMessage := Base.F_GetLastWordInString(__POUNAME());
END_IF

IF NOT _DispatchValid() THEN
	RETURN;
ELSE
	_BuildCommandStringNoArgs();
	
	IF iBufferSend <> 0 AND __QUERYINTERFACE(iBufferSend, testIBufferSend) THEN
		iBufferSend.AddObject(RefObject := ZaberCommand);
	END_IF
END_IF
END_METHOD

METHOD get_ictrl_afcff_ss
IF ZaberStatus.ComponentStatus.iLastCommand <> 0 THEN
	ZaberStatus.ComponentStatus.iLastCommand.P_CommandStatus.LastCommandMessage := Base.F_GetLastWordInString(__POUNAME());
END_IF

IF NOT _DispatchValid() THEN
	RETURN;
ELSE
	_BuildCommandStringNoArgs();
	
	IF iBufferSend <> 0 AND __QUERYINTERFACE(iBufferSend, testIBufferSend) THEN
		iBufferSend.AddObject(RefObject := ZaberCommand);
	END_IF
END_IF
END_METHOD

METHOD get_ictrl_afcff_ss_max
IF ZaberStatus.ComponentStatus.iLastCommand <> 0 THEN
	ZaberStatus.ComponentStatus.iLastCommand.P_CommandStatus.LastCommandMessage := Base.F_GetLastWordInString(__POUNAME());
END_IF

IF NOT _DispatchValid() THEN
	RETURN;
ELSE
	_BuildCommandStringNoArgs();
	
	IF iBufferSend <> 0 AND __QUERYINTERFACE(iBufferSend, testIBufferSend) THEN
		iBufferSend.AddObject(RefObject := ZaberCommand);
	END_IF
END_IF
END_METHOD

METHOD get_ictrl_delay
IF ZaberStatus.ComponentStatus.iLastCommand <> 0 THEN
	ZaberStatus.ComponentStatus.iLastCommand.P_CommandStatus.LastCommandMessage := Base.F_GetLastWordInString(__POUNAME());
END_IF

IF NOT _DispatchValid() THEN
	RETURN;
ELSE
	_BuildCommandStringNoArgs();
	
	IF iBufferSend <> 0 AND __QUERYINTERFACE(iBufferSend, testIBufferSend) THEN
		iBufferSend.AddObject(RefObject := ZaberCommand);
	END_IF
END_IF
END_METHOD

METHOD get_ictrl_ff_kd
IF ZaberStatus.ComponentStatus.iLastCommand <> 0 THEN
	ZaberStatus.ComponentStatus.iLastCommand.P_CommandStatus.LastCommandMessage := Base.F_GetLastWordInString(__POUNAME());
END_IF

IF NOT _DispatchValid() THEN
	RETURN;
ELSE
	_BuildCommandStringNoArgs();
	
	IF iBufferSend <> 0 AND __QUERYINTERFACE(iBufferSend, testIBufferSend) THEN
		iBufferSend.AddObject(RefObject := ZaberCommand);
	END_IF
END_IF
END_METHOD

METHOD get_ictrl_ff_kp
IF ZaberStatus.ComponentStatus.iLastCommand <> 0 THEN
	ZaberStatus.ComponentStatus.iLastCommand.P_CommandStatus.LastCommandMessage := Base.F_GetLastWordInString(__POUNAME());
END_IF

IF NOT _DispatchValid() THEN
	RETURN;
ELSE
	_BuildCommandStringNoArgs();
	
	IF iBufferSend <> 0 AND __QUERYINTERFACE(iBufferSend, testIBufferSend) THEN
		iBufferSend.AddObject(RefObject := ZaberCommand);
	END_IF
END_IF
END_METHOD

METHOD get_ictrl_gain_coldmult
IF ZaberStatus.ComponentStatus.iLastCommand <> 0 THEN
	ZaberStatus.ComponentStatus.iLastCommand.P_CommandStatus.LastCommandMessage := Base.F_GetLastWordInString(__POUNAME());
END_IF

IF NOT _DispatchValid() THEN
	RETURN;
ELSE
	_BuildCommandStringNoArgs();
	
	IF iBufferSend <> 0 AND __QUERYINTERFACE(iBufferSend, testIBufferSend) THEN
		iBufferSend.AddObject(RefObject := ZaberCommand);
	END_IF
END_IF
END_METHOD

METHOD get_ictrl_period
IF ZaberStatus.ComponentStatus.iLastCommand <> 0 THEN
	ZaberStatus.ComponentStatus.iLastCommand.P_CommandStatus.LastCommandMessage := Base.F_GetLastWordInString(__POUNAME());
END_IF

IF NOT _DispatchValid() THEN
	RETURN;
ELSE
	_BuildCommandStringNoArgs();
	
	IF iBufferSend <> 0 AND __QUERYINTERFACE(iBufferSend, testIBufferSend) THEN
		iBufferSend.AddObject(RefObject := ZaberCommand);
	END_IF
END_IF
END_METHOD

METHOD get_ictrl_pi_ki
IF ZaberStatus.ComponentStatus.iLastCommand <> 0 THEN
	ZaberStatus.ComponentStatus.iLastCommand.P_CommandStatus.LastCommandMessage := Base.F_GetLastWordInString(__POUNAME());
END_IF

IF NOT _DispatchValid() THEN
	RETURN;
ELSE
	_BuildCommandStringNoArgs();
	
	IF iBufferSend <> 0 AND __QUERYINTERFACE(iBufferSend, testIBufferSend) THEN
		iBufferSend.AddObject(RefObject := ZaberCommand);
	END_IF
END_IF
END_METHOD

METHOD get_ictrl_pi_kp
IF ZaberStatus.ComponentStatus.iLastCommand <> 0 THEN
	ZaberStatus.ComponentStatus.iLastCommand.P_CommandStatus.LastCommandMessage := Base.F_GetLastWordInString(__POUNAME());
END_IF

IF NOT _DispatchValid() THEN
	RETURN;
ELSE
	_BuildCommandStringNoArgs();
	
	IF iBufferSend <> 0 AND __QUERYINTERFACE(iBufferSend, testIBufferSend) THEN
		iBufferSend.AddObject(RefObject := ZaberCommand);
	END_IF
END_IF
END_METHOD

METHOD get_ictrl_type
IF ZaberStatus.ComponentStatus.iLastCommand <> 0 THEN
	ZaberStatus.ComponentStatus.iLastCommand.P_CommandStatus.LastCommandMessage := Base.F_GetLastWordInString(__POUNAME());
END_IF

IF NOT _DispatchValid() THEN
	RETURN;
ELSE
	_BuildCommandStringNoArgs();
	
	IF iBufferSend <> 0 AND __QUERYINTERFACE(iBufferSend, testIBufferSend) THEN
		iBufferSend.AddObject(RefObject := ZaberCommand);
	END_IF
END_IF
END_METHOD

METHOD get_io_ai_1_fc
IF ZaberStatus.ComponentStatus.iLastCommand <> 0 THEN
	ZaberStatus.ComponentStatus.iLastCommand.P_CommandStatus.LastCommandMessage := Base.F_GetLastWordInString(__POUNAME());
END_IF

IF NOT _DispatchValid() THEN
	RETURN;
ELSE
	_BuildCommandStringNoArgs();
	
	IF iBufferSend <> 0 AND __QUERYINTERFACE(iBufferSend, testIBufferSend) THEN
		iBufferSend.AddObject(RefObject := ZaberCommand);
	END_IF
END_IF
END_METHOD

METHOD get_io_ai_2_fc
IF ZaberStatus.ComponentStatus.iLastCommand <> 0 THEN
	ZaberStatus.ComponentStatus.iLastCommand.P_CommandStatus.LastCommandMessage := Base.F_GetLastWordInString(__POUNAME());
END_IF

IF NOT _DispatchValid() THEN
	RETURN;
ELSE
	_BuildCommandStringNoArgs();
	
	IF iBufferSend <> 0 AND __QUERYINTERFACE(iBufferSend, testIBufferSend) THEN
		iBufferSend.AddObject(RefObject := ZaberCommand);
	END_IF
END_IF
END_METHOD

METHOD get_io_ai_3_fc
IF ZaberStatus.ComponentStatus.iLastCommand <> 0 THEN
	ZaberStatus.ComponentStatus.iLastCommand.P_CommandStatus.LastCommandMessage := Base.F_GetLastWordInString(__POUNAME());
END_IF

IF NOT _DispatchValid() THEN
	RETURN;
ELSE
	_BuildCommandStringNoArgs();
	
	IF iBufferSend <> 0 AND __QUERYINTERFACE(iBufferSend, testIBufferSend) THEN
		iBufferSend.AddObject(RefObject := ZaberCommand);
	END_IF
END_IF
END_METHOD

METHOD get_io_ai_4_fc
IF ZaberStatus.ComponentStatus.iLastCommand <> 0 THEN
	ZaberStatus.ComponentStatus.iLastCommand.P_CommandStatus.LastCommandMessage := Base.F_GetLastWordInString(__POUNAME());
END_IF

IF NOT _DispatchValid() THEN
	RETURN;
ELSE
	_BuildCommandStringNoArgs();
	
	IF iBufferSend <> 0 AND __QUERYINTERFACE(iBufferSend, testIBufferSend) THEN
		iBufferSend.AddObject(RefObject := ZaberCommand);
	END_IF
END_IF
END_METHOD

METHOD get_io_di_port
IF ZaberStatus.ComponentStatus.iLastCommand <> 0 THEN
	ZaberStatus.ComponentStatus.iLastCommand.P_CommandStatus.LastCommandMessage := Base.F_GetLastWordInString(__POUNAME());
END_IF

IF NOT _DispatchValid() THEN
	RETURN;
ELSE
	_BuildCommandStringNoArgs();
	
	IF iBufferSend <> 0 AND __QUERYINTERFACE(iBufferSend, testIBufferSend) THEN
		iBufferSend.AddObject(RefObject := ZaberCommand);
	END_IF
END_IF
END_METHOD

METHOD get_io_do_port
IF ZaberStatus.ComponentStatus.iLastCommand <> 0 THEN
	ZaberStatus.ComponentStatus.iLastCommand.P_CommandStatus.LastCommandMessage := Base.F_GetLastWordInString(__POUNAME());
END_IF

IF NOT _DispatchValid() THEN
	RETURN;
ELSE
	_BuildCommandStringNoArgs();
	
	IF iBufferSend <> 0 AND __QUERYINTERFACE(iBufferSend, testIBufferSend) THEN
		iBufferSend.AddObject(RefObject := ZaberCommand);
	END_IF
END_IF
END_METHOD

METHOD get_knob_dir
IF ZaberStatus.ComponentStatus.iLastCommand <> 0 THEN
	ZaberStatus.ComponentStatus.iLastCommand.P_CommandStatus.LastCommandMessage := Base.F_GetLastWordInString(__POUNAME());
END_IF

IF NOT _DispatchValid() THEN
	RETURN;
ELSE
	_BuildCommandStringNoArgs();
	
	IF iBufferSend <> 0 AND __QUERYINTERFACE(iBufferSend, testIBufferSend) THEN
		iBufferSend.AddObject(RefObject := ZaberCommand);
	END_IF
END_IF
END_METHOD

METHOD get_knob_distance
IF ZaberStatus.ComponentStatus.iLastCommand <> 0 THEN
	ZaberStatus.ComponentStatus.iLastCommand.P_CommandStatus.LastCommandMessage := Base.F_GetLastWordInString(__POUNAME());
END_IF

IF NOT _DispatchValid() THEN
	RETURN;
ELSE
	_BuildCommandStringNoArgs();
	
	IF iBufferSend <> 0 AND __QUERYINTERFACE(iBufferSend, testIBufferSend) THEN
		iBufferSend.AddObject(RefObject := ZaberCommand);
	END_IF
END_IF
END_METHOD

METHOD get_knob_enable
IF ZaberStatus.ComponentStatus.iLastCommand <> 0 THEN
	ZaberStatus.ComponentStatus.iLastCommand.P_CommandStatus.LastCommandMessage := Base.F_GetLastWordInString(__POUNAME());
END_IF

IF NOT _DispatchValid() THEN
	RETURN;
ELSE
	_BuildCommandStringNoArgs();
	
	IF iBufferSend <> 0 AND __QUERYINTERFACE(iBufferSend, testIBufferSend) THEN
		iBufferSend.AddObject(RefObject := ZaberCommand);
	END_IF
END_IF
END_METHOD

METHOD get_knob_maxspeed
IF ZaberStatus.ComponentStatus.iLastCommand <> 0 THEN
	ZaberStatus.ComponentStatus.iLastCommand.P_CommandStatus.LastCommandMessage := Base.F_GetLastWordInString(__POUNAME());
END_IF

IF NOT _DispatchValid() THEN
	RETURN;
ELSE
	_BuildCommandStringNoArgs();
	
	IF iBufferSend <> 0 AND __QUERYINTERFACE(iBufferSend, testIBufferSend) THEN
		iBufferSend.AddObject(RefObject := ZaberCommand);
	END_IF
END_IF
END_METHOD

METHOD get_knob_mode
IF ZaberStatus.ComponentStatus.iLastCommand <> 0 THEN
	ZaberStatus.ComponentStatus.iLastCommand.P_CommandStatus.LastCommandMessage := Base.F_GetLastWordInString(__POUNAME());
END_IF

IF NOT _DispatchValid() THEN
	RETURN;
ELSE
	_BuildCommandStringNoArgs();
	
	IF iBufferSend <> 0 AND __QUERYINTERFACE(iBufferSend, testIBufferSend) THEN
		iBufferSend.AddObject(RefObject := ZaberCommand);
	END_IF
END_IF
END_METHOD

METHOD get_knob_speedprofile
IF ZaberStatus.ComponentStatus.iLastCommand <> 0 THEN
	ZaberStatus.ComponentStatus.iLastCommand.P_CommandStatus.LastCommandMessage := Base.F_GetLastWordInString(__POUNAME());
END_IF

IF NOT _DispatchValid() THEN
	RETURN;
ELSE
	_BuildCommandStringNoArgs();
	
	IF iBufferSend <> 0 AND __QUERYINTERFACE(iBufferSend, testIBufferSend) THEN
		iBufferSend.AddObject(RefObject := ZaberCommand);
	END_IF
END_IF
END_METHOD

METHOD get_limit_approach_maxspeed
IF ZaberStatus.ComponentStatus.iLastCommand <> 0 THEN
	ZaberStatus.ComponentStatus.iLastCommand.P_CommandStatus.LastCommandMessage := Base.F_GetLastWordInString(__POUNAME());
END_IF

IF NOT _DispatchValid() THEN
	RETURN;
ELSE
	_BuildCommandStringNoArgs();
	
	IF iBufferSend <> 0 AND __QUERYINTERFACE(iBufferSend, testIBufferSend) THEN
		iBufferSend.AddObject(RefObject := ZaberCommand);
	END_IF
END_IF
END_METHOD

METHOD get_limit_detect_decelonly
IF ZaberStatus.ComponentStatus.iLastCommand <> 0 THEN
	ZaberStatus.ComponentStatus.iLastCommand.P_CommandStatus.LastCommandMessage := Base.F_GetLastWordInString(__POUNAME());
END_IF

IF NOT _DispatchValid() THEN
	RETURN;
ELSE
	_BuildCommandStringNoArgs();
	
	IF iBufferSend <> 0 AND __QUERYINTERFACE(iBufferSend, testIBufferSend) THEN
		iBufferSend.AddObject(RefObject := ZaberCommand);
	END_IF
END_IF
END_METHOD

METHOD get_limit_detect_maxspeed
IF ZaberStatus.ComponentStatus.iLastCommand <> 0 THEN
	ZaberStatus.ComponentStatus.iLastCommand.P_CommandStatus.LastCommandMessage := Base.F_GetLastWordInString(__POUNAME());
END_IF

IF NOT _DispatchValid() THEN
	RETURN;
ELSE
	_BuildCommandStringNoArgs();
	
	IF iBufferSend <> 0 AND __QUERYINTERFACE(iBufferSend, testIBufferSend) THEN
		iBufferSend.AddObject(RefObject := ZaberCommand);
	END_IF
END_IF
END_METHOD

METHOD get_limit_home_action
IF ZaberStatus.ComponentStatus.iLastCommand <> 0 THEN
	ZaberStatus.ComponentStatus.iLastCommand.P_CommandStatus.LastCommandMessage := Base.F_GetLastWordInString(__POUNAME());
END_IF

IF NOT _DispatchValid() THEN
	RETURN;
ELSE
	_BuildCommandStringNoArgs();
	
	IF iBufferSend <> 0 AND __QUERYINTERFACE(iBufferSend, testIBufferSend) THEN
		iBufferSend.AddObject(RefObject := ZaberCommand);
	END_IF
END_IF
END_METHOD

METHOD get_limit_home_bidirectional
IF ZaberStatus.ComponentStatus.iLastCommand <> 0 THEN
	ZaberStatus.ComponentStatus.iLastCommand.P_CommandStatus.LastCommandMessage := Base.F_GetLastWordInString(__POUNAME());
END_IF

IF NOT _DispatchValid() THEN
	RETURN;
ELSE
	_BuildCommandStringNoArgs();
	
	IF iBufferSend <> 0 AND __QUERYINTERFACE(iBufferSend, testIBufferSend) THEN
		iBufferSend.AddObject(RefObject := ZaberCommand);
	END_IF
END_IF
END_METHOD

METHOD get_limit_home_edge
IF ZaberStatus.ComponentStatus.iLastCommand <> 0 THEN
	ZaberStatus.ComponentStatus.iLastCommand.P_CommandStatus.LastCommandMessage := Base.F_GetLastWordInString(__POUNAME());
END_IF

IF NOT _DispatchValid() THEN
	RETURN;
ELSE
	_BuildCommandStringNoArgs();
	
	IF iBufferSend <> 0 AND __QUERYINTERFACE(iBufferSend, testIBufferSend) THEN
		iBufferSend.AddObject(RefObject := ZaberCommand);
	END_IF
END_IF
END_METHOD

METHOD get_limit_home_offset
IF ZaberStatus.ComponentStatus.iLastCommand <> 0 THEN
	ZaberStatus.ComponentStatus.iLastCommand.P_CommandStatus.LastCommandMessage := Base.F_GetLastWordInString(__POUNAME());
END_IF

IF NOT _DispatchValid() THEN
	RETURN;
ELSE
	_BuildCommandStringNoArgs();
	
	IF iBufferSend <> 0 AND __QUERYINTERFACE(iBufferSend, testIBufferSend) THEN
		iBufferSend.AddObject(RefObject := ZaberCommand);
	END_IF
END_IF
END_METHOD

METHOD get_limit_home_posupdate
IF ZaberStatus.ComponentStatus.iLastCommand <> 0 THEN
	ZaberStatus.ComponentStatus.iLastCommand.P_CommandStatus.LastCommandMessage := Base.F_GetLastWordInString(__POUNAME());
END_IF

IF NOT _DispatchValid() THEN
	RETURN;
ELSE
	_BuildCommandStringNoArgs();
	
	IF iBufferSend <> 0 AND __QUERYINTERFACE(iBufferSend, testIBufferSend) THEN
		iBufferSend.AddObject(RefObject := ZaberCommand);
	END_IF
END_IF
END_METHOD

METHOD get_limit_home_preset
IF ZaberStatus.ComponentStatus.iLastCommand <> 0 THEN
	ZaberStatus.ComponentStatus.iLastCommand.P_CommandStatus.LastCommandMessage := Base.F_GetLastWordInString(__POUNAME());
END_IF

IF NOT _DispatchValid() THEN
	RETURN;
ELSE
	_BuildCommandStringNoArgs();
	
	IF iBufferSend <> 0 AND __QUERYINTERFACE(iBufferSend, testIBufferSend) THEN
		iBufferSend.AddObject(RefObject := ZaberCommand);
	END_IF
END_IF
END_METHOD

METHOD get_limit_home_source
IF ZaberStatus.ComponentStatus.iLastCommand <> 0 THEN
	ZaberStatus.ComponentStatus.iLastCommand.P_CommandStatus.LastCommandMessage := Base.F_GetLastWordInString(__POUNAME());
END_IF

IF NOT _DispatchValid() THEN
	RETURN;
ELSE
	_BuildCommandStringNoArgs();
	
	IF iBufferSend <> 0 AND __QUERYINTERFACE(iBufferSend, testIBufferSend) THEN
		iBufferSend.AddObject(RefObject := ZaberCommand);
	END_IF
END_IF
END_METHOD

METHOD get_limit_home_state
IF ZaberStatus.ComponentStatus.iLastCommand <> 0 THEN
	ZaberStatus.ComponentStatus.iLastCommand.P_CommandStatus.LastCommandMessage := Base.F_GetLastWordInString(__POUNAME());
END_IF

IF NOT _DispatchValid() THEN
	RETURN;
ELSE
	_BuildCommandStringNoArgs();
	
	IF iBufferSend <> 0 AND __QUERYINTERFACE(iBufferSend, testIBufferSend) THEN
		iBufferSend.AddObject(RefObject := ZaberCommand);
	END_IF
END_IF
END_METHOD

METHOD get_limit_home_triggered
IF ZaberStatus.ComponentStatus.iLastCommand <> 0 THEN
	ZaberStatus.ComponentStatus.iLastCommand.P_CommandStatus.LastCommandMessage := Base.F_GetLastWordInString(__POUNAME());
END_IF

IF NOT _DispatchValid() THEN
	RETURN;
ELSE
	_BuildCommandStringNoArgs();
	
	IF iBufferSend <> 0 AND __QUERYINTERFACE(iBufferSend, testIBufferSend) THEN
		iBufferSend.AddObject(RefObject := ZaberCommand);
	END_IF
END_IF
END_METHOD

METHOD get_limit_home_tune
IF ZaberStatus.ComponentStatus.iLastCommand <> 0 THEN
	ZaberStatus.ComponentStatus.iLastCommand.P_CommandStatus.LastCommandMessage := Base.F_GetLastWordInString(__POUNAME());
END_IF

IF NOT _DispatchValid() THEN
	RETURN;
ELSE
	_BuildCommandStringNoArgs();
	
	IF iBufferSend <> 0 AND __QUERYINTERFACE(iBufferSend, testIBufferSend) THEN
		iBufferSend.AddObject(RefObject := ZaberCommand);
	END_IF
END_IF
END_METHOD

METHOD get_limit_home_type
IF ZaberStatus.ComponentStatus.iLastCommand <> 0 THEN
	ZaberStatus.ComponentStatus.iLastCommand.P_CommandStatus.LastCommandMessage := Base.F_GetLastWordInString(__POUNAME());
END_IF

IF NOT _DispatchValid() THEN
	RETURN;
ELSE
	_BuildCommandStringNoArgs();
	
	IF iBufferSend <> 0 AND __QUERYINTERFACE(iBufferSend, testIBufferSend) THEN
		iBufferSend.AddObject(RefObject := ZaberCommand);
	END_IF
END_IF
END_METHOD

METHOD get_limit_home_width
IF ZaberStatus.ComponentStatus.iLastCommand <> 0 THEN
	ZaberStatus.ComponentStatus.iLastCommand.P_CommandStatus.LastCommandMessage := Base.F_GetLastWordInString(__POUNAME());
END_IF

IF NOT _DispatchValid() THEN
	RETURN;
ELSE
	_BuildCommandStringNoArgs();
	
	IF iBufferSend <> 0 AND __QUERYINTERFACE(iBufferSend, testIBufferSend) THEN
		iBufferSend.AddObject(RefObject := ZaberCommand);
	END_IF
END_IF
END_METHOD

METHOD get_limit_max
IF ZaberStatus.ComponentStatus.iLastCommand <> 0 THEN
	ZaberStatus.ComponentStatus.iLastCommand.P_CommandStatus.LastCommandMessage := Base.F_GetLastWordInString(__POUNAME());
END_IF

IF NOT _DispatchValid() THEN
	RETURN;
ELSE
	_BuildCommandStringNoArgs();
	
	IF iBufferSend <> 0 AND __QUERYINTERFACE(iBufferSend, testIBufferSend) THEN
		iBufferSend.AddObject(RefObject := ZaberCommand);
	END_IF
END_IF
END_METHOD

METHOD get_limit_min
IF ZaberStatus.ComponentStatus.iLastCommand <> 0 THEN
	ZaberStatus.ComponentStatus.iLastCommand.P_CommandStatus.LastCommandMessage := Base.F_GetLastWordInString(__POUNAME());
END_IF

IF NOT _DispatchValid() THEN
	RETURN;
ELSE
	_BuildCommandStringNoArgs();
	
	IF iBufferSend <> 0 AND __QUERYINTERFACE(iBufferSend, testIBufferSend) THEN
		iBufferSend.AddObject(RefObject := ZaberCommand);
	END_IF
END_IF
END_METHOD

METHOD get_limit_range_mode
IF ZaberStatus.ComponentStatus.iLastCommand <> 0 THEN
	ZaberStatus.ComponentStatus.iLastCommand.P_CommandStatus.LastCommandMessage := Base.F_GetLastWordInString(__POUNAME());
END_IF

IF NOT _DispatchValid() THEN
	RETURN;
ELSE
	_BuildCommandStringNoArgs();
	
	IF iBufferSend <> 0 AND __QUERYINTERFACE(iBufferSend, testIBufferSend) THEN
		iBufferSend.AddObject(RefObject := ZaberCommand);
	END_IF
END_IF
END_METHOD

METHOD get_lockstep_numgroups
IF ZaberStatus.ComponentStatus.iLastCommand <> 0 THEN
	ZaberStatus.ComponentStatus.iLastCommand.P_CommandStatus.LastCommandMessage := Base.F_GetLastWordInString(__POUNAME());
END_IF

IF NOT _DispatchValid() THEN
	RETURN;
ELSE
	_BuildCommandStringNoArgs();
	
	IF iBufferSend <> 0 AND __QUERYINTERFACE(iBufferSend, testIBufferSend) THEN
		iBufferSend.AddObject(RefObject := ZaberCommand);
	END_IF
END_IF
END_METHOD

METHOD get_maxspeed
IF ZaberStatus.ComponentStatus.iLastCommand <> 0 THEN
	ZaberStatus.ComponentStatus.iLastCommand.P_CommandStatus.LastCommandMessage := Base.F_GetLastWordInString(__POUNAME());
END_IF

IF NOT _DispatchValid() THEN
	RETURN;
ELSE
	_BuildCommandStringNoArgs();
	
	IF iBufferSend <> 0 AND __QUERYINTERFACE(iBufferSend, testIBufferSend) THEN
		iBufferSend.AddObject(RefObject := ZaberCommand);
	END_IF
END_IF
END_METHOD

METHOD get_motion_accel_ramptime
IF ZaberStatus.ComponentStatus.iLastCommand <> 0 THEN
	ZaberStatus.ComponentStatus.iLastCommand.P_CommandStatus.LastCommandMessage := Base.F_GetLastWordInString(__POUNAME());
END_IF

IF NOT _DispatchValid() THEN
	RETURN;
ELSE
	_BuildCommandStringNoArgs();
	
	IF iBufferSend <> 0 AND __QUERYINTERFACE(iBufferSend, testIBufferSend) THEN
		iBufferSend.AddObject(RefObject := ZaberCommand);
	END_IF
END_IF
END_METHOD

METHOD get_motion_accelonly
IF ZaberStatus.ComponentStatus.iLastCommand <> 0 THEN
	ZaberStatus.ComponentStatus.iLastCommand.P_CommandStatus.LastCommandMessage := Base.F_GetLastWordInString(__POUNAME());
END_IF

IF NOT _DispatchValid() THEN
	RETURN;
ELSE
	_BuildCommandStringNoArgs();
	
	IF iBufferSend <> 0 AND __QUERYINTERFACE(iBufferSend, testIBufferSend) THEN
		iBufferSend.AddObject(RefObject := ZaberCommand);
	END_IF
END_IF
END_METHOD

METHOD get_motion_busy
IF ZaberStatus.ComponentStatus.iLastCommand <> 0 THEN
	ZaberStatus.ComponentStatus.iLastCommand.P_CommandStatus.LastCommandMessage := Base.F_GetLastWordInString(__POUNAME());
END_IF

IF NOT _DispatchValid() THEN
	RETURN;
ELSE
	_BuildCommandStringNoArgs();
	
	IF iBufferSend <> 0 AND __QUERYINTERFACE(iBufferSend, testIBufferSend) THEN
		iBufferSend.AddObject(RefObject := ZaberCommand);
	END_IF
END_IF
END_METHOD

METHOD get_motion_decelonly
IF ZaberStatus.ComponentStatus.iLastCommand <> 0 THEN
	ZaberStatus.ComponentStatus.iLastCommand.P_CommandStatus.LastCommandMessage := Base.F_GetLastWordInString(__POUNAME());
END_IF

IF NOT _DispatchValid() THEN
	RETURN;
ELSE
	_BuildCommandStringNoArgs();
	
	IF iBufferSend <> 0 AND __QUERYINTERFACE(iBufferSend, testIBufferSend) THEN
		iBufferSend.AddObject(RefObject := ZaberCommand);
	END_IF
END_IF
END_METHOD

METHOD get_motion_index_dist
IF ZaberStatus.ComponentStatus.iLastCommand <> 0 THEN
	ZaberStatus.ComponentStatus.iLastCommand.P_CommandStatus.LastCommandMessage := Base.F_GetLastWordInString(__POUNAME());
END_IF

IF NOT _DispatchValid() THEN
	RETURN;
ELSE
	_BuildCommandStringNoArgs();
	
	IF iBufferSend <> 0 AND __QUERYINTERFACE(iBufferSend, testIBufferSend) THEN
		iBufferSend.AddObject(RefObject := ZaberCommand);
	END_IF
END_IF
END_METHOD

METHOD get_motion_index_num
IF ZaberStatus.ComponentStatus.iLastCommand <> 0 THEN
	ZaberStatus.ComponentStatus.iLastCommand.P_CommandStatus.LastCommandMessage := Base.F_GetLastWordInString(__POUNAME());
END_IF

IF NOT _DispatchValid() THEN
	RETURN;
ELSE
	_BuildCommandStringNoArgs();
	
	IF iBufferSend <> 0 AND __QUERYINTERFACE(iBufferSend, testIBufferSend) THEN
		iBufferSend.AddObject(RefObject := ZaberCommand);
	END_IF
END_IF
END_METHOD

METHOD get_motion_tracking_ai
IF ZaberStatus.ComponentStatus.iLastCommand <> 0 THEN
	ZaberStatus.ComponentStatus.iLastCommand.P_CommandStatus.LastCommandMessage := Base.F_GetLastWordInString(__POUNAME());
END_IF

IF NOT _DispatchValid() THEN
	RETURN;
ELSE
	_BuildCommandStringNoArgs();
	
	IF iBufferSend <> 0 AND __QUERYINTERFACE(iBufferSend, testIBufferSend) THEN
		iBufferSend.AddObject(RefObject := ZaberCommand);
	END_IF
END_IF
END_METHOD

METHOD get_motion_tracking_dir
IF ZaberStatus.ComponentStatus.iLastCommand <> 0 THEN
	ZaberStatus.ComponentStatus.iLastCommand.P_CommandStatus.LastCommandMessage := Base.F_GetLastWordInString(__POUNAME());
END_IF

IF NOT _DispatchValid() THEN
	RETURN;
ELSE
	_BuildCommandStringNoArgs();
	
	IF iBufferSend <> 0 AND __QUERYINTERFACE(iBufferSend, testIBufferSend) THEN
		iBufferSend.AddObject(RefObject := ZaberCommand);
	END_IF
END_IF
END_METHOD

METHOD get_motion_tracking_ki
IF ZaberStatus.ComponentStatus.iLastCommand <> 0 THEN
	ZaberStatus.ComponentStatus.iLastCommand.P_CommandStatus.LastCommandMessage := Base.F_GetLastWordInString(__POUNAME());
END_IF

IF NOT _DispatchValid() THEN
	RETURN;
ELSE
	_BuildCommandStringNoArgs();
	
	IF iBufferSend <> 0 AND __QUERYINTERFACE(iBufferSend, testIBufferSend) THEN
		iBufferSend.AddObject(RefObject := ZaberCommand);
	END_IF
END_IF
END_METHOD

METHOD get_motion_tracking_kp
IF ZaberStatus.ComponentStatus.iLastCommand <> 0 THEN
	ZaberStatus.ComponentStatus.iLastCommand.P_CommandStatus.LastCommandMessage := Base.F_GetLastWordInString(__POUNAME());
END_IF

IF NOT _DispatchValid() THEN
	RETURN;
ELSE
	_BuildCommandStringNoArgs();
	
	IF iBufferSend <> 0 AND __QUERYINTERFACE(iBufferSend, testIBufferSend) THEN
		iBufferSend.AddObject(RefObject := ZaberCommand);
	END_IF
END_IF
END_METHOD

METHOD get_motion_tracking_limit_max
IF ZaberStatus.ComponentStatus.iLastCommand <> 0 THEN
	ZaberStatus.ComponentStatus.iLastCommand.P_CommandStatus.LastCommandMessage := Base.F_GetLastWordInString(__POUNAME());
END_IF

IF NOT _DispatchValid() THEN
	RETURN;
ELSE
	_BuildCommandStringNoArgs();
	
	IF iBufferSend <> 0 AND __QUERYINTERFACE(iBufferSend, testIBufferSend) THEN
		iBufferSend.AddObject(RefObject := ZaberCommand);
	END_IF
END_IF
END_METHOD

METHOD get_motion_tracking_limit_min
IF ZaberStatus.ComponentStatus.iLastCommand <> 0 THEN
	ZaberStatus.ComponentStatus.iLastCommand.P_CommandStatus.LastCommandMessage := Base.F_GetLastWordInString(__POUNAME());
END_IF

IF NOT _DispatchValid() THEN
	RETURN;
ELSE
	_BuildCommandStringNoArgs();
	
	IF iBufferSend <> 0 AND __QUERYINTERFACE(iBufferSend, testIBufferSend) THEN
		iBufferSend.AddObject(RefObject := ZaberCommand);
	END_IF
END_IF
END_METHOD

METHOD get_motion_tracking_scan_dir
IF ZaberStatus.ComponentStatus.iLastCommand <> 0 THEN
	ZaberStatus.ComponentStatus.iLastCommand.P_CommandStatus.LastCommandMessage := Base.F_GetLastWordInString(__POUNAME());
END_IF

IF NOT _DispatchValid() THEN
	RETURN;
ELSE
	_BuildCommandStringNoArgs();
	
	IF iBufferSend <> 0 AND __QUERYINTERFACE(iBufferSend, testIBufferSend) THEN
		iBufferSend.AddObject(RefObject := ZaberCommand);
	END_IF
END_IF
END_METHOD

METHOD get_motion_tracking_scan_maxspeed
IF ZaberStatus.ComponentStatus.iLastCommand <> 0 THEN
	ZaberStatus.ComponentStatus.iLastCommand.P_CommandStatus.LastCommandMessage := Base.F_GetLastWordInString(__POUNAME());
END_IF

IF NOT _DispatchValid() THEN
	RETURN;
ELSE
	_BuildCommandStringNoArgs();
	
	IF iBufferSend <> 0 AND __QUERYINTERFACE(iBufferSend, testIBufferSend) THEN
		iBufferSend.AddObject(RefObject := ZaberCommand);
	END_IF
END_IF
END_METHOD

METHOD get_motion_tracking_scan_offset
IF ZaberStatus.ComponentStatus.iLastCommand <> 0 THEN
	ZaberStatus.ComponentStatus.iLastCommand.P_CommandStatus.LastCommandMessage := Base.F_GetLastWordInString(__POUNAME());
END_IF

IF NOT _DispatchValid() THEN
	RETURN;
ELSE
	_BuildCommandStringNoArgs();
	
	IF iBufferSend <> 0 AND __QUERYINTERFACE(iBufferSend, testIBufferSend) THEN
		iBufferSend.AddObject(RefObject := ZaberCommand);
	END_IF
END_IF
END_METHOD

METHOD get_motion_tracking_scan_period
IF ZaberStatus.ComponentStatus.iLastCommand <> 0 THEN
	ZaberStatus.ComponentStatus.iLastCommand.P_CommandStatus.LastCommandMessage := Base.F_GetLastWordInString(__POUNAME());
END_IF

IF NOT _DispatchValid() THEN
	RETURN;
ELSE
	_BuildCommandStringNoArgs();
	
	IF iBufferSend <> 0 AND __QUERYINTERFACE(iBufferSend, testIBufferSend) THEN
		iBufferSend.AddObject(RefObject := ZaberCommand);
	END_IF
END_IF
END_METHOD

METHOD get_motion_tracking_scan_signal_valid_delay
IF ZaberStatus.ComponentStatus.iLastCommand <> 0 THEN
	ZaberStatus.ComponentStatus.iLastCommand.P_CommandStatus.LastCommandMessage := Base.F_GetLastWordInString(__POUNAME());
END_IF

IF NOT _DispatchValid() THEN
	RETURN;
ELSE
	_BuildCommandStringNoArgs();
	
	IF iBufferSend <> 0 AND __QUERYINTERFACE(iBufferSend, testIBufferSend) THEN
		iBufferSend.AddObject(RefObject := ZaberCommand);
	END_IF
END_IF
END_METHOD

METHOD get_motion_tracking_scan_tolerance
IF ZaberStatus.ComponentStatus.iLastCommand <> 0 THEN
	ZaberStatus.ComponentStatus.iLastCommand.P_CommandStatus.LastCommandMessage := Base.F_GetLastWordInString(__POUNAME());
END_IF

IF NOT _DispatchValid() THEN
	RETURN;
ELSE
	_BuildCommandStringNoArgs();
	
	IF iBufferSend <> 0 AND __QUERYINTERFACE(iBufferSend, testIBufferSend) THEN
		iBufferSend.AddObject(RefObject := ZaberCommand);
	END_IF
END_IF
END_METHOD

METHOD get_motion_tracking_setpoint
IF ZaberStatus.ComponentStatus.iLastCommand <> 0 THEN
	ZaberStatus.ComponentStatus.iLastCommand.P_CommandStatus.LastCommandMessage := Base.F_GetLastWordInString(__POUNAME());
END_IF

IF NOT _DispatchValid() THEN
	RETURN;
ELSE
	_BuildCommandStringNoArgs();
	
	IF iBufferSend <> 0 AND __QUERYINTERFACE(iBufferSend, testIBufferSend) THEN
		iBufferSend.AddObject(RefObject := ZaberCommand);
	END_IF
END_IF
END_METHOD

METHOD get_motion_tracking_settle_period
IF ZaberStatus.ComponentStatus.iLastCommand <> 0 THEN
	ZaberStatus.ComponentStatus.iLastCommand.P_CommandStatus.LastCommandMessage := Base.F_GetLastWordInString(__POUNAME());
END_IF

IF NOT _DispatchValid() THEN
	RETURN;
ELSE
	_BuildCommandStringNoArgs();
	
	IF iBufferSend <> 0 AND __QUERYINTERFACE(iBufferSend, testIBufferSend) THEN
		iBufferSend.AddObject(RefObject := ZaberCommand);
	END_IF
END_IF
END_METHOD

METHOD get_motion_tracking_settle_tolerance
IF ZaberStatus.ComponentStatus.iLastCommand <> 0 THEN
	ZaberStatus.ComponentStatus.iLastCommand.P_CommandStatus.LastCommandMessage := Base.F_GetLastWordInString(__POUNAME());
END_IF

IF NOT _DispatchValid() THEN
	RETURN;
ELSE
	_BuildCommandStringNoArgs();
	
	IF iBufferSend <> 0 AND __QUERYINTERFACE(iBufferSend, testIBufferSend) THEN
		iBufferSend.AddObject(RefObject := ZaberCommand);
	END_IF
END_IF
END_METHOD

METHOD get_motion_tracking_settle_tolerance_met
IF ZaberStatus.ComponentStatus.iLastCommand <> 0 THEN
	ZaberStatus.ComponentStatus.iLastCommand.P_CommandStatus.LastCommandMessage := Base.F_GetLastWordInString(__POUNAME());
END_IF

IF NOT _DispatchValid() THEN
	RETURN;
ELSE
	_BuildCommandStringNoArgs();
	
	IF iBufferSend <> 0 AND __QUERYINTERFACE(iBufferSend, testIBufferSend) THEN
		iBufferSend.AddObject(RefObject := ZaberCommand);
	END_IF
END_IF
END_METHOD

METHOD get_motion_tracking_settled
IF ZaberStatus.ComponentStatus.iLastCommand <> 0 THEN
	ZaberStatus.ComponentStatus.iLastCommand.P_CommandStatus.LastCommandMessage := Base.F_GetLastWordInString(__POUNAME());
END_IF

IF NOT _DispatchValid() THEN
	RETURN;
ELSE
	_BuildCommandStringNoArgs();
	
	IF iBufferSend <> 0 AND __QUERYINTERFACE(iBufferSend, testIBufferSend) THEN
		iBufferSend.AddObject(RefObject := ZaberCommand);
	END_IF
END_IF
END_METHOD

METHOD get_motion_tracking_signal_valid_di
IF ZaberStatus.ComponentStatus.iLastCommand <> 0 THEN
	ZaberStatus.ComponentStatus.iLastCommand.P_CommandStatus.LastCommandMessage := Base.F_GetLastWordInString(__POUNAME());
END_IF

IF NOT _DispatchValid() THEN
	RETURN;
ELSE
	_BuildCommandStringNoArgs();
	
	IF iBufferSend <> 0 AND __QUERYINTERFACE(iBufferSend, testIBufferSend) THEN
		iBufferSend.AddObject(RefObject := ZaberCommand);
	END_IF
END_IF
END_METHOD

METHOD get_motor_current_max
IF ZaberStatus.ComponentStatus.iLastCommand <> 0 THEN
	ZaberStatus.ComponentStatus.iLastCommand.P_CommandStatus.LastCommandMessage := Base.F_GetLastWordInString(__POUNAME());
END_IF

IF NOT _DispatchValid() THEN
	RETURN;
ELSE
	_BuildCommandStringNoArgs();
	
	IF iBufferSend <> 0 AND __QUERYINTERFACE(iBufferSend, testIBufferSend) THEN
		iBufferSend.AddObject(RefObject := ZaberCommand);
	END_IF
END_IF
END_METHOD

METHOD get_motor_inductance
IF ZaberStatus.ComponentStatus.iLastCommand <> 0 THEN
	ZaberStatus.ComponentStatus.iLastCommand.P_CommandStatus.LastCommandMessage := Base.F_GetLastWordInString(__POUNAME());
END_IF

IF NOT _DispatchValid() THEN
	RETURN;
ELSE
	_BuildCommandStringNoArgs();
	
	IF iBufferSend <> 0 AND __QUERYINTERFACE(iBufferSend, testIBufferSend) THEN
		iBufferSend.AddObject(RefObject := ZaberCommand);
	END_IF
END_IF
END_METHOD

METHOD get_motor_ke
IF ZaberStatus.ComponentStatus.iLastCommand <> 0 THEN
	ZaberStatus.ComponentStatus.iLastCommand.P_CommandStatus.LastCommandMessage := Base.F_GetLastWordInString(__POUNAME());
END_IF

IF NOT _DispatchValid() THEN
	RETURN;
ELSE
	_BuildCommandStringNoArgs();
	
	IF iBufferSend <> 0 AND __QUERYINTERFACE(iBufferSend, testIBufferSend) THEN
		iBufferSend.AddObject(RefObject := ZaberCommand);
	END_IF
END_IF
END_METHOD

METHOD get_motor_phase
IF ZaberStatus.ComponentStatus.iLastCommand <> 0 THEN
	ZaberStatus.ComponentStatus.iLastCommand.P_CommandStatus.LastCommandMessage := Base.F_GetLastWordInString(__POUNAME());
END_IF

IF NOT _DispatchValid() THEN
	RETURN;
ELSE
	_BuildCommandStringNoArgs();
	
	IF iBufferSend <> 0 AND __QUERYINTERFACE(iBufferSend, testIBufferSend) THEN
		iBufferSend.AddObject(RefObject := ZaberCommand);
	END_IF
END_IF
END_METHOD

METHOD get_motor_phase_ratio_div1
IF ZaberStatus.ComponentStatus.iLastCommand <> 0 THEN
	ZaberStatus.ComponentStatus.iLastCommand.P_CommandStatus.LastCommandMessage := Base.F_GetLastWordInString(__POUNAME());
END_IF

IF NOT _DispatchValid() THEN
	RETURN;
ELSE
	_BuildCommandStringNoArgs();
	
	IF iBufferSend <> 0 AND __QUERYINTERFACE(iBufferSend, testIBufferSend) THEN
		iBufferSend.AddObject(RefObject := ZaberCommand);
	END_IF
END_IF
END_METHOD

METHOD get_motor_phase_ratio_div2
IF ZaberStatus.ComponentStatus.iLastCommand <> 0 THEN
	ZaberStatus.ComponentStatus.iLastCommand.P_CommandStatus.LastCommandMessage := Base.F_GetLastWordInString(__POUNAME());
END_IF

IF NOT _DispatchValid() THEN
	RETURN;
ELSE
	_BuildCommandStringNoArgs();
	
	IF iBufferSend <> 0 AND __QUERYINTERFACE(iBufferSend, testIBufferSend) THEN
		iBufferSend.AddObject(RefObject := ZaberCommand);
	END_IF
END_IF
END_METHOD

METHOD get_motor_phase_ratio_mult
IF ZaberStatus.ComponentStatus.iLastCommand <> 0 THEN
	ZaberStatus.ComponentStatus.iLastCommand.P_CommandStatus.LastCommandMessage := Base.F_GetLastWordInString(__POUNAME());
END_IF

IF NOT _DispatchValid() THEN
	RETURN;
ELSE
	_BuildCommandStringNoArgs();
	
	IF iBufferSend <> 0 AND __QUERYINTERFACE(iBufferSend, testIBufferSend) THEN
		iBufferSend.AddObject(RefObject := ZaberCommand);
	END_IF
END_IF
END_METHOD

METHOD get_motor_resistance
IF ZaberStatus.ComponentStatus.iLastCommand <> 0 THEN
	ZaberStatus.ComponentStatus.iLastCommand.P_CommandStatus.LastCommandMessage := Base.F_GetLastWordInString(__POUNAME());
END_IF

IF NOT _DispatchValid() THEN
	RETURN;
ELSE
	_BuildCommandStringNoArgs();
	
	IF iBufferSend <> 0 AND __QUERYINTERFACE(iBufferSend, testIBufferSend) THEN
		iBufferSend.AddObject(RefObject := ZaberCommand);
	END_IF
END_IF
END_METHOD

METHOD get_parking_state
IF ZaberStatus.ComponentStatus.iLastCommand <> 0 THEN
	ZaberStatus.ComponentStatus.iLastCommand.P_CommandStatus.LastCommandMessage := Base.F_GetLastWordInString(__POUNAME());
END_IF

IF NOT _DispatchValid() THEN
	RETURN;
ELSE
	_BuildCommandStringNoArgs();
	
	IF iBufferSend <> 0 AND __QUERYINTERFACE(iBufferSend, testIBufferSend) THEN
		iBufferSend.AddObject(RefObject := ZaberCommand);
	END_IF
END_IF
END_METHOD

METHOD get_peripheral_hw_modified
IF ZaberStatus.ComponentStatus.iLastCommand <> 0 THEN
	ZaberStatus.ComponentStatus.iLastCommand.P_CommandStatus.LastCommandMessage := Base.F_GetLastWordInString(__POUNAME());
END_IF

IF NOT _DispatchValid() THEN
	RETURN;
ELSE
	_BuildCommandStringNoArgs();
	
	IF iBufferSend <> 0 AND __QUERYINTERFACE(iBufferSend, testIBufferSend) THEN
		iBufferSend.AddObject(RefObject := ZaberCommand);
	END_IF
END_IF
END_METHOD

METHOD get_peripheral_id
IF ZaberStatus.ComponentStatus.iLastCommand <> 0 THEN
	ZaberStatus.ComponentStatus.iLastCommand.P_CommandStatus.LastCommandMessage := Base.F_GetLastWordInString(__POUNAME());
END_IF

IF NOT _DispatchValid() THEN
	RETURN;
ELSE
	_BuildCommandStringNoArgs();
	
	IF iBufferSend <> 0 AND __QUERYINTERFACE(iBufferSend, testIBufferSend) THEN
		iBufferSend.AddObject(RefObject := ZaberCommand);
	END_IF
END_IF
END_METHOD

METHOD get_peripheral_id_pending
IF ZaberStatus.ComponentStatus.iLastCommand <> 0 THEN
	ZaberStatus.ComponentStatus.iLastCommand.P_CommandStatus.LastCommandMessage := Base.F_GetLastWordInString(__POUNAME());
END_IF

IF NOT _DispatchValid() THEN
	RETURN;
ELSE
	_BuildCommandStringNoArgs();
	
	IF iBufferSend <> 0 AND __QUERYINTERFACE(iBufferSend, testIBufferSend) THEN
		iBufferSend.AddObject(RefObject := ZaberCommand);
	END_IF
END_IF
END_METHOD

METHOD get_peripheral_serial
IF ZaberStatus.ComponentStatus.iLastCommand <> 0 THEN
	ZaberStatus.ComponentStatus.iLastCommand.P_CommandStatus.LastCommandMessage := Base.F_GetLastWordInString(__POUNAME());
END_IF

IF NOT _DispatchValid() THEN
	RETURN;
ELSE
	_BuildCommandStringNoArgs();
	
	IF iBufferSend <> 0 AND __QUERYINTERFACE(iBufferSend, testIBufferSend) THEN
		iBufferSend.AddObject(RefObject := ZaberCommand);
	END_IF
END_IF
END_METHOD

METHOD get_peripheral_serial_pending
IF ZaberStatus.ComponentStatus.iLastCommand <> 0 THEN
	ZaberStatus.ComponentStatus.iLastCommand.P_CommandStatus.LastCommandMessage := Base.F_GetLastWordInString(__POUNAME());
END_IF

IF NOT _DispatchValid() THEN
	RETURN;
ELSE
	_BuildCommandStringNoArgs();
	
	IF iBufferSend <> 0 AND __QUERYINTERFACE(iBufferSend, testIBufferSend) THEN
		iBufferSend.AddObject(RefObject := ZaberCommand);
	END_IF
END_IF
END_METHOD

METHOD get_pos
IF ZaberStatus.ComponentStatus.iLastCommand <> 0 THEN
	ZaberStatus.ComponentStatus.iLastCommand.P_CommandStatus.LastCommandMessage := Base.F_GetLastWordInString(__POUNAME());
END_IF

IF NOT _DispatchValid() THEN
	RETURN;
ELSE
	_BuildCommandStringNoArgs();
	
	IF iBufferSend <> 0 AND __QUERYINTERFACE(iBufferSend, testIBufferSend) THEN
		iBufferSend.AddObject(RefObject := ZaberCommand);
	END_IF
END_IF
END_METHOD

METHOD get_pvt_numseqs
IF ZaberStatus.ComponentStatus.iLastCommand <> 0 THEN
	ZaberStatus.ComponentStatus.iLastCommand.P_CommandStatus.LastCommandMessage := Base.F_GetLastWordInString(__POUNAME());
END_IF

IF NOT _DispatchValid() THEN
	RETURN;
ELSE
	_BuildCommandStringNoArgs();
	
	IF iBufferSend <> 0 AND __QUERYINTERFACE(iBufferSend, testIBufferSend) THEN
		iBufferSend.AddObject(RefObject := ZaberCommand);
	END_IF
END_IF
END_METHOD

METHOD get_resolution
IF ZaberStatus.ComponentStatus.iLastCommand <> 0 THEN
	ZaberStatus.ComponentStatus.iLastCommand.P_CommandStatus.LastCommandMessage := Base.F_GetLastWordInString(__POUNAME());
END_IF

IF NOT _DispatchValid() THEN
	RETURN;
ELSE
	_BuildCommandStringNoArgs();
	
	IF iBufferSend <> 0 AND __QUERYINTERFACE(iBufferSend, testIBufferSend) THEN
		iBufferSend.AddObject(RefObject := ZaberCommand);
	END_IF
END_IF
END_METHOD

METHOD get_scope_channel_size
IF ZaberStatus.ComponentStatus.iLastCommand <> 0 THEN
	ZaberStatus.ComponentStatus.iLastCommand.P_CommandStatus.LastCommandMessage := Base.F_GetLastWordInString(__POUNAME());
END_IF

IF NOT _DispatchValid() THEN
	RETURN;
ELSE
	_BuildCommandStringNoArgs();
	
	IF iBufferSend <> 0 AND __QUERYINTERFACE(iBufferSend, testIBufferSend) THEN
		iBufferSend.AddObject(RefObject := ZaberCommand);
	END_IF
END_IF
END_METHOD

METHOD get_scope_channel_size_max
IF ZaberStatus.ComponentStatus.iLastCommand <> 0 THEN
	ZaberStatus.ComponentStatus.iLastCommand.P_CommandStatus.LastCommandMessage := Base.F_GetLastWordInString(__POUNAME());
END_IF

IF NOT _DispatchValid() THEN
	RETURN;
ELSE
	_BuildCommandStringNoArgs();
	
	IF iBufferSend <> 0 AND __QUERYINTERFACE(iBufferSend, testIBufferSend) THEN
		iBufferSend.AddObject(RefObject := ZaberCommand);
	END_IF
END_IF
END_METHOD

METHOD get_scope_delay
IF ZaberStatus.ComponentStatus.iLastCommand <> 0 THEN
	ZaberStatus.ComponentStatus.iLastCommand.P_CommandStatus.LastCommandMessage := Base.F_GetLastWordInString(__POUNAME());
END_IF

IF NOT _DispatchValid() THEN
	RETURN;
ELSE
	_BuildCommandStringNoArgs();
	
	IF iBufferSend <> 0 AND __QUERYINTERFACE(iBufferSend, testIBufferSend) THEN
		iBufferSend.AddObject(RefObject := ZaberCommand);
	END_IF
END_IF
END_METHOD

METHOD get_scope_numchannels
IF ZaberStatus.ComponentStatus.iLastCommand <> 0 THEN
	ZaberStatus.ComponentStatus.iLastCommand.P_CommandStatus.LastCommandMessage := Base.F_GetLastWordInString(__POUNAME());
END_IF

IF NOT _DispatchValid() THEN
	RETURN;
ELSE
	_BuildCommandStringNoArgs();
	
	IF iBufferSend <> 0 AND __QUERYINTERFACE(iBufferSend, testIBufferSend) THEN
		iBufferSend.AddObject(RefObject := ZaberCommand);
	END_IF
END_IF
END_METHOD

METHOD get_scope_timebase
IF ZaberStatus.ComponentStatus.iLastCommand <> 0 THEN
	ZaberStatus.ComponentStatus.iLastCommand.P_CommandStatus.LastCommandMessage := Base.F_GetLastWordInString(__POUNAME());
END_IF

IF NOT _DispatchValid() THEN
	RETURN;
ELSE
	_BuildCommandStringNoArgs();
	
	IF iBufferSend <> 0 AND __QUERYINTERFACE(iBufferSend, testIBufferSend) THEN
		iBufferSend.AddObject(RefObject := ZaberCommand);
	END_IF
END_IF
END_METHOD

METHOD get_stream_numbufs
IF ZaberStatus.ComponentStatus.iLastCommand <> 0 THEN
	ZaberStatus.ComponentStatus.iLastCommand.P_CommandStatus.LastCommandMessage := Base.F_GetLastWordInString(__POUNAME());
END_IF

IF NOT _DispatchValid() THEN
	RETURN;
ELSE
	_BuildCommandStringNoArgs();
	
	IF iBufferSend <> 0 AND __QUERYINTERFACE(iBufferSend, testIBufferSend) THEN
		iBufferSend.AddObject(RefObject := ZaberCommand);
	END_IF
END_IF
END_METHOD

METHOD get_stream_numstreams
IF ZaberStatus.ComponentStatus.iLastCommand <> 0 THEN
	ZaberStatus.ComponentStatus.iLastCommand.P_CommandStatus.LastCommandMessage := Base.F_GetLastWordInString(__POUNAME());
END_IF

IF NOT _DispatchValid() THEN
	RETURN;
ELSE
	_BuildCommandStringNoArgs();
	
	IF iBufferSend <> 0 AND __QUERYINTERFACE(iBufferSend, testIBufferSend) THEN
		iBufferSend.AddObject(RefObject := ZaberCommand);
	END_IF
END_IF
END_METHOD

METHOD get_system_access
IF ZaberStatus.ComponentStatus.iLastCommand <> 0 THEN
	ZaberStatus.ComponentStatus.iLastCommand.P_CommandStatus.LastCommandMessage := Base.F_GetLastWordInString(__POUNAME());
END_IF

IF NOT _DispatchValid() THEN
	RETURN;
ELSE
	_BuildCommandStringNoArgs();
	
	IF iBufferSend <> 0 AND __QUERYINTERFACE(iBufferSend, testIBufferSend) THEN
		iBufferSend.AddObject(RefObject := ZaberCommand);
	END_IF
END_IF
END_METHOD

METHOD get_system_axiscount
IF ZaberStatus.ComponentStatus.iLastCommand <> 0 THEN
	ZaberStatus.ComponentStatus.iLastCommand.P_CommandStatus.LastCommandMessage := Base.F_GetLastWordInString(__POUNAME());
END_IF

IF NOT _DispatchValid() THEN
	RETURN;
ELSE
	_BuildCommandStringNoArgs();
	
	IF iBufferSend <> 0 AND __QUERYINTERFACE(iBufferSend, testIBufferSend) THEN
		iBufferSend.AddObject(RefObject := ZaberCommand);
	END_IF
END_IF
END_METHOD

METHOD get_system_current_max
IF ZaberStatus.ComponentStatus.iLastCommand <> 0 THEN
	ZaberStatus.ComponentStatus.iLastCommand.P_CommandStatus.LastCommandMessage := Base.F_GetLastWordInString(__POUNAME());
END_IF

IF NOT _DispatchValid() THEN
	RETURN;
ELSE
	_BuildCommandStringNoArgs();
	
	IF iBufferSend <> 0 AND __QUERYINTERFACE(iBufferSend, testIBufferSend) THEN
		iBufferSend.AddObject(RefObject := ZaberCommand);
	END_IF
END_IF
END_METHOD

METHOD get_system_led_enable
IF ZaberStatus.ComponentStatus.iLastCommand <> 0 THEN
	ZaberStatus.ComponentStatus.iLastCommand.P_CommandStatus.LastCommandMessage := Base.F_GetLastWordInString(__POUNAME());
END_IF

IF NOT _DispatchValid() THEN
	RETURN;
ELSE
	_BuildCommandStringNoArgs();
	
	IF iBufferSend <> 0 AND __QUERYINTERFACE(iBufferSend, testIBufferSend) THEN
		iBufferSend.AddObject(RefObject := ZaberCommand);
	END_IF
END_IF
END_METHOD

METHOD get_system_serial
IF ZaberStatus.ComponentStatus.iLastCommand <> 0 THEN
	ZaberStatus.ComponentStatus.iLastCommand.P_CommandStatus.LastCommandMessage := Base.F_GetLastWordInString(__POUNAME());
END_IF

IF NOT _DispatchValid() THEN
	RETURN;
ELSE
	_BuildCommandStringNoArgs();
	
	IF iBufferSend <> 0 AND __QUERYINTERFACE(iBufferSend, testIBufferSend) THEN
		iBufferSend.AddObject(RefObject := ZaberCommand);
	END_IF
END_IF
END_METHOD

METHOD get_system_temperature
IF ZaberStatus.ComponentStatus.iLastCommand <> 0 THEN
	ZaberStatus.ComponentStatus.iLastCommand.P_CommandStatus.LastCommandMessage := Base.F_GetLastWordInString(__POUNAME());
END_IF

IF NOT _DispatchValid() THEN
	RETURN;
ELSE
	_BuildCommandStringNoArgs();
	
	IF iBufferSend <> 0 AND __QUERYINTERFACE(iBufferSend, testIBufferSend) THEN
		iBufferSend.AddObject(RefObject := ZaberCommand);
	END_IF
END_IF
END_METHOD

METHOD get_system_uptime
IF ZaberStatus.ComponentStatus.iLastCommand <> 0 THEN
	ZaberStatus.ComponentStatus.iLastCommand.P_CommandStatus.LastCommandMessage := Base.F_GetLastWordInString(__POUNAME());
END_IF

IF NOT _DispatchValid() THEN
	RETURN;
ELSE
	_BuildCommandStringNoArgs();
	
	IF iBufferSend <> 0 AND __QUERYINTERFACE(iBufferSend, testIBufferSend) THEN
		iBufferSend.AddObject(RefObject := ZaberCommand);
	END_IF
END_IF
END_METHOD

METHOD get_system_voltage
IF ZaberStatus.ComponentStatus.iLastCommand <> 0 THEN
	ZaberStatus.ComponentStatus.iLastCommand.P_CommandStatus.LastCommandMessage := Base.F_GetLastWordInString(__POUNAME());
END_IF

IF NOT _DispatchValid() THEN
	RETURN;
ELSE
	_BuildCommandStringNoArgs();
	
	IF iBufferSend <> 0 AND __QUERYINTERFACE(iBufferSend, testIBufferSend) THEN
		iBufferSend.AddObject(RefObject := ZaberCommand);
	END_IF
END_IF
END_METHOD

METHOD get_trigger_numactions
IF ZaberStatus.ComponentStatus.iLastCommand <> 0 THEN
	ZaberStatus.ComponentStatus.iLastCommand.P_CommandStatus.LastCommandMessage := Base.F_GetLastWordInString(__POUNAME());
END_IF

IF NOT _DispatchValid() THEN
	RETURN;
ELSE
	_BuildCommandStringNoArgs();
	
	IF iBufferSend <> 0 AND __QUERYINTERFACE(iBufferSend, testIBufferSend) THEN
		iBufferSend.AddObject(RefObject := ZaberCommand);
	END_IF
END_IF
END_METHOD

METHOD get_trigger_numtriggers
IF ZaberStatus.ComponentStatus.iLastCommand <> 0 THEN
	ZaberStatus.ComponentStatus.iLastCommand.P_CommandStatus.LastCommandMessage := Base.F_GetLastWordInString(__POUNAME());
END_IF

IF NOT _DispatchValid() THEN
	RETURN;
ELSE
	_BuildCommandStringNoArgs();
	
	IF iBufferSend <> 0 AND __QUERYINTERFACE(iBufferSend, testIBufferSend) THEN
		iBufferSend.AddObject(RefObject := ZaberCommand);
	END_IF
END_IF
END_METHOD

METHOD get_user_data_0
IF ZaberStatus.ComponentStatus.iLastCommand <> 0 THEN
	ZaberStatus.ComponentStatus.iLastCommand.P_CommandStatus.LastCommandMessage := Base.F_GetLastWordInString(__POUNAME());
END_IF

IF NOT _DispatchValid() THEN
	RETURN;
ELSE
	_BuildCommandStringNoArgs();
	
	IF iBufferSend <> 0 AND __QUERYINTERFACE(iBufferSend, testIBufferSend) THEN
		iBufferSend.AddObject(RefObject := ZaberCommand);
	END_IF
END_IF
END_METHOD

METHOD get_user_data_1
IF ZaberStatus.ComponentStatus.iLastCommand <> 0 THEN
	ZaberStatus.ComponentStatus.iLastCommand.P_CommandStatus.LastCommandMessage := Base.F_GetLastWordInString(__POUNAME());
END_IF

IF NOT _DispatchValid() THEN
	RETURN;
ELSE
	_BuildCommandStringNoArgs();
	
	IF iBufferSend <> 0 AND __QUERYINTERFACE(iBufferSend, testIBufferSend) THEN
		iBufferSend.AddObject(RefObject := ZaberCommand);
	END_IF
END_IF
END_METHOD

METHOD get_user_data_10
IF ZaberStatus.ComponentStatus.iLastCommand <> 0 THEN
	ZaberStatus.ComponentStatus.iLastCommand.P_CommandStatus.LastCommandMessage := Base.F_GetLastWordInString(__POUNAME());
END_IF

IF NOT _DispatchValid() THEN
	RETURN;
ELSE
	_BuildCommandStringNoArgs();
	
	IF iBufferSend <> 0 AND __QUERYINTERFACE(iBufferSend, testIBufferSend) THEN
		iBufferSend.AddObject(RefObject := ZaberCommand);
	END_IF
END_IF
END_METHOD

METHOD get_user_data_11
IF ZaberStatus.ComponentStatus.iLastCommand <> 0 THEN
	ZaberStatus.ComponentStatus.iLastCommand.P_CommandStatus.LastCommandMessage := Base.F_GetLastWordInString(__POUNAME());
END_IF

IF NOT _DispatchValid() THEN
	RETURN;
ELSE
	_BuildCommandStringNoArgs();
	
	IF iBufferSend <> 0 AND __QUERYINTERFACE(iBufferSend, testIBufferSend) THEN
		iBufferSend.AddObject(RefObject := ZaberCommand);
	END_IF
END_IF
END_METHOD

METHOD get_user_data_12
IF ZaberStatus.ComponentStatus.iLastCommand <> 0 THEN
	ZaberStatus.ComponentStatus.iLastCommand.P_CommandStatus.LastCommandMessage := Base.F_GetLastWordInString(__POUNAME());
END_IF

IF NOT _DispatchValid() THEN
	RETURN;
ELSE
	_BuildCommandStringNoArgs();
	
	IF iBufferSend <> 0 AND __QUERYINTERFACE(iBufferSend, testIBufferSend) THEN
		iBufferSend.AddObject(RefObject := ZaberCommand);
	END_IF
END_IF
END_METHOD

METHOD get_user_data_13
IF ZaberStatus.ComponentStatus.iLastCommand <> 0 THEN
	ZaberStatus.ComponentStatus.iLastCommand.P_CommandStatus.LastCommandMessage := Base.F_GetLastWordInString(__POUNAME());
END_IF

IF NOT _DispatchValid() THEN
	RETURN;
ELSE
	_BuildCommandStringNoArgs();
	
	IF iBufferSend <> 0 AND __QUERYINTERFACE(iBufferSend, testIBufferSend) THEN
		iBufferSend.AddObject(RefObject := ZaberCommand);
	END_IF
END_IF
END_METHOD

METHOD get_user_data_14
IF ZaberStatus.ComponentStatus.iLastCommand <> 0 THEN
	ZaberStatus.ComponentStatus.iLastCommand.P_CommandStatus.LastCommandMessage := Base.F_GetLastWordInString(__POUNAME());
END_IF

IF NOT _DispatchValid() THEN
	RETURN;
ELSE
	_BuildCommandStringNoArgs();
	
	IF iBufferSend <> 0 AND __QUERYINTERFACE(iBufferSend, testIBufferSend) THEN
		iBufferSend.AddObject(RefObject := ZaberCommand);
	END_IF
END_IF
END_METHOD

METHOD get_user_data_15
IF ZaberStatus.ComponentStatus.iLastCommand <> 0 THEN
	ZaberStatus.ComponentStatus.iLastCommand.P_CommandStatus.LastCommandMessage := Base.F_GetLastWordInString(__POUNAME());
END_IF

IF NOT _DispatchValid() THEN
	RETURN;
ELSE
	_BuildCommandStringNoArgs();
	
	IF iBufferSend <> 0 AND __QUERYINTERFACE(iBufferSend, testIBufferSend) THEN
		iBufferSend.AddObject(RefObject := ZaberCommand);
	END_IF
END_IF
END_METHOD

METHOD get_user_data_2
IF ZaberStatus.ComponentStatus.iLastCommand <> 0 THEN
	ZaberStatus.ComponentStatus.iLastCommand.P_CommandStatus.LastCommandMessage := Base.F_GetLastWordInString(__POUNAME());
END_IF

IF NOT _DispatchValid() THEN
	RETURN;
ELSE
	_BuildCommandStringNoArgs();
	
	IF iBufferSend <> 0 AND __QUERYINTERFACE(iBufferSend, testIBufferSend) THEN
		iBufferSend.AddObject(RefObject := ZaberCommand);
	END_IF
END_IF
END_METHOD

METHOD get_user_data_3
IF ZaberStatus.ComponentStatus.iLastCommand <> 0 THEN
	ZaberStatus.ComponentStatus.iLastCommand.P_CommandStatus.LastCommandMessage := Base.F_GetLastWordInString(__POUNAME());
END_IF

IF NOT _DispatchValid() THEN
	RETURN;
ELSE
	_BuildCommandStringNoArgs();
	
	IF iBufferSend <> 0 AND __QUERYINTERFACE(iBufferSend, testIBufferSend) THEN
		iBufferSend.AddObject(RefObject := ZaberCommand);
	END_IF
END_IF
END_METHOD

METHOD get_user_data_4
IF ZaberStatus.ComponentStatus.iLastCommand <> 0 THEN
	ZaberStatus.ComponentStatus.iLastCommand.P_CommandStatus.LastCommandMessage := Base.F_GetLastWordInString(__POUNAME());
END_IF

IF NOT _DispatchValid() THEN
	RETURN;
ELSE
	_BuildCommandStringNoArgs();
	
	IF iBufferSend <> 0 AND __QUERYINTERFACE(iBufferSend, testIBufferSend) THEN
		iBufferSend.AddObject(RefObject := ZaberCommand);
	END_IF
END_IF
END_METHOD

METHOD get_user_data_5
IF ZaberStatus.ComponentStatus.iLastCommand <> 0 THEN
	ZaberStatus.ComponentStatus.iLastCommand.P_CommandStatus.LastCommandMessage := Base.F_GetLastWordInString(__POUNAME());
END_IF

IF NOT _DispatchValid() THEN
	RETURN;
ELSE
	_BuildCommandStringNoArgs();
	
	IF iBufferSend <> 0 AND __QUERYINTERFACE(iBufferSend, testIBufferSend) THEN
		iBufferSend.AddObject(RefObject := ZaberCommand);
	END_IF
END_IF
END_METHOD

METHOD get_user_data_6
IF ZaberStatus.ComponentStatus.iLastCommand <> 0 THEN
	ZaberStatus.ComponentStatus.iLastCommand.P_CommandStatus.LastCommandMessage := Base.F_GetLastWordInString(__POUNAME());
END_IF

IF NOT _DispatchValid() THEN
	RETURN;
ELSE
	_BuildCommandStringNoArgs();
	
	IF iBufferSend <> 0 AND __QUERYINTERFACE(iBufferSend, testIBufferSend) THEN
		iBufferSend.AddObject(RefObject := ZaberCommand);
	END_IF
END_IF
END_METHOD

METHOD get_user_data_7
IF ZaberStatus.ComponentStatus.iLastCommand <> 0 THEN
	ZaberStatus.ComponentStatus.iLastCommand.P_CommandStatus.LastCommandMessage := Base.F_GetLastWordInString(__POUNAME());
END_IF

IF NOT _DispatchValid() THEN
	RETURN;
ELSE
	_BuildCommandStringNoArgs();
	
	IF iBufferSend <> 0 AND __QUERYINTERFACE(iBufferSend, testIBufferSend) THEN
		iBufferSend.AddObject(RefObject := ZaberCommand);
	END_IF
END_IF
END_METHOD

METHOD get_user_data_8
IF ZaberStatus.ComponentStatus.iLastCommand <> 0 THEN
	ZaberStatus.ComponentStatus.iLastCommand.P_CommandStatus.LastCommandMessage := Base.F_GetLastWordInString(__POUNAME());
END_IF

IF NOT _DispatchValid() THEN
	RETURN;
ELSE
	_BuildCommandStringNoArgs();
	
	IF iBufferSend <> 0 AND __QUERYINTERFACE(iBufferSend, testIBufferSend) THEN
		iBufferSend.AddObject(RefObject := ZaberCommand);
	END_IF
END_IF
END_METHOD

METHOD get_user_data_9
IF ZaberStatus.ComponentStatus.iLastCommand <> 0 THEN
	ZaberStatus.ComponentStatus.iLastCommand.P_CommandStatus.LastCommandMessage := Base.F_GetLastWordInString(__POUNAME());
END_IF

IF NOT _DispatchValid() THEN
	RETURN;
ELSE
	_BuildCommandStringNoArgs();
	
	IF iBufferSend <> 0 AND __QUERYINTERFACE(iBufferSend, testIBufferSend) THEN
		iBufferSend.AddObject(RefObject := ZaberCommand);
	END_IF
END_IF
END_METHOD

METHOD get_user_vdata_0
IF ZaberStatus.ComponentStatus.iLastCommand <> 0 THEN
	ZaberStatus.ComponentStatus.iLastCommand.P_CommandStatus.LastCommandMessage := Base.F_GetLastWordInString(__POUNAME());
END_IF

IF NOT _DispatchValid() THEN
	RETURN;
ELSE
	_BuildCommandStringNoArgs();
	
	IF iBufferSend <> 0 AND __QUERYINTERFACE(iBufferSend, testIBufferSend) THEN
		iBufferSend.AddObject(RefObject := ZaberCommand);
	END_IF
END_IF
END_METHOD

METHOD get_user_vdata_1
IF ZaberStatus.ComponentStatus.iLastCommand <> 0 THEN
	ZaberStatus.ComponentStatus.iLastCommand.P_CommandStatus.LastCommandMessage := Base.F_GetLastWordInString(__POUNAME());
END_IF

IF NOT _DispatchValid() THEN
	RETURN;
ELSE
	_BuildCommandStringNoArgs();
	
	IF iBufferSend <> 0 AND __QUERYINTERFACE(iBufferSend, testIBufferSend) THEN
		iBufferSend.AddObject(RefObject := ZaberCommand);
	END_IF
END_IF
END_METHOD

METHOD get_user_vdata_2
IF ZaberStatus.ComponentStatus.iLastCommand <> 0 THEN
	ZaberStatus.ComponentStatus.iLastCommand.P_CommandStatus.LastCommandMessage := Base.F_GetLastWordInString(__POUNAME());
END_IF

IF NOT _DispatchValid() THEN
	RETURN;
ELSE
	_BuildCommandStringNoArgs();
	
	IF iBufferSend <> 0 AND __QUERYINTERFACE(iBufferSend, testIBufferSend) THEN
		iBufferSend.AddObject(RefObject := ZaberCommand);
	END_IF
END_IF
END_METHOD

METHOD get_user_vdata_3
IF ZaberStatus.ComponentStatus.iLastCommand <> 0 THEN
	ZaberStatus.ComponentStatus.iLastCommand.P_CommandStatus.LastCommandMessage := Base.F_GetLastWordInString(__POUNAME());
END_IF

IF NOT _DispatchValid() THEN
	RETURN;
ELSE
	_BuildCommandStringNoArgs();
	
	IF iBufferSend <> 0 AND __QUERYINTERFACE(iBufferSend, testIBufferSend) THEN
		iBufferSend.AddObject(RefObject := ZaberCommand);
	END_IF
END_IF
END_METHOD

METHOD get_vel
IF ZaberStatus.ComponentStatus.iLastCommand <> 0 THEN
	ZaberStatus.ComponentStatus.iLastCommand.P_CommandStatus.LastCommandMessage := Base.F_GetLastWordInString(__POUNAME());
END_IF

IF NOT _DispatchValid() THEN
	RETURN;
ELSE
	_BuildCommandStringNoArgs();
	
	IF iBufferSend <> 0 AND __QUERYINTERFACE(iBufferSend, testIBufferSend) THEN
		iBufferSend.AddObject(RefObject := ZaberCommand);
	END_IF
END_IF
END_METHOD

METHOD get_version
IF ZaberStatus.ComponentStatus.iLastCommand <> 0 THEN
	ZaberStatus.ComponentStatus.iLastCommand.P_CommandStatus.LastCommandMessage := Base.F_GetLastWordInString(__POUNAME());
END_IF

IF NOT _DispatchValid() THEN
	RETURN;
ELSE
	_BuildCommandStringNoArgs();
	
	IF iBufferSend <> 0 AND __QUERYINTERFACE(iBufferSend, testIBufferSend) THEN
		iBufferSend.AddObject(RefObject := ZaberCommand);
	END_IF
END_IF
END_METHOD

METHOD get_version_build
IF ZaberStatus.ComponentStatus.iLastCommand <> 0 THEN
	ZaberStatus.ComponentStatus.iLastCommand.P_CommandStatus.LastCommandMessage := Base.F_GetLastWordInString(__POUNAME());
END_IF

IF NOT _DispatchValid() THEN
	RETURN;
ELSE
	_BuildCommandStringNoArgs();
	
	IF iBufferSend <> 0 AND __QUERYINTERFACE(iBufferSend, testIBufferSend) THEN
		iBufferSend.AddObject(RefObject := ZaberCommand);
	END_IF
END_IF
END_METHOD

METHOD home
IF ZaberStatus.ComponentStatus.iLastCommand <> 0 THEN
	ZaberStatus.ComponentStatus.iLastCommand.P_CommandStatus.LastCommandMessage := Base.F_GetLastWordInString(__POUNAME());
END_IF

IF NOT _DispatchValid() THEN
	RETURN;
ELSE
	_BuildCommandStringNoArgs();
	
	IF iBufferSend <> 0 AND __QUERYINTERFACE(iBufferSend, testIBufferSend) THEN
		iBufferSend.AddObject(RefObject := ZaberCommand);
	END_IF
END_IF
END_METHOD

METHOD io_get_ai
IF ZaberStatus.ComponentStatus.iLastCommand <> 0 THEN
	ZaberStatus.ComponentStatus.iLastCommand.P_CommandStatus.LastCommandMessage := Base.F_GetLastWordInString(__POUNAME());
END_IF

IF NOT _DispatchValid() THEN
	RETURN;
ELSE
	_BuildCommandStringNoArgs();
	
	IF iBufferSend <> 0 AND __QUERYINTERFACE(iBufferSend, testIBufferSend) THEN
		iBufferSend.AddObject(RefObject := ZaberCommand);
	END_IF
END_IF
END_METHOD

METHOD io_get_ao
IF ZaberStatus.ComponentStatus.iLastCommand <> 0 THEN
	ZaberStatus.ComponentStatus.iLastCommand.P_CommandStatus.LastCommandMessage := Base.F_GetLastWordInString(__POUNAME());
END_IF

IF NOT _DispatchValid() THEN
	RETURN;
ELSE
	_BuildCommandStringNoArgs();
	
	IF iBufferSend <> 0 AND __QUERYINTERFACE(iBufferSend, testIBufferSend) THEN
		iBufferSend.AddObject(RefObject := ZaberCommand);
	END_IF
END_IF
END_METHOD

METHOD io_get_di
IF ZaberStatus.ComponentStatus.iLastCommand <> 0 THEN
	ZaberStatus.ComponentStatus.iLastCommand.P_CommandStatus.LastCommandMessage := Base.F_GetLastWordInString(__POUNAME());
END_IF

IF NOT _DispatchValid() THEN
	RETURN;
ELSE
	_BuildCommandStringNoArgs();
	
	IF iBufferSend <> 0 AND __QUERYINTERFACE(iBufferSend, testIBufferSend) THEN
		iBufferSend.AddObject(RefObject := ZaberCommand);
	END_IF
END_IF
END_METHOD

METHOD io_get_do
IF ZaberStatus.ComponentStatus.iLastCommand <> 0 THEN
	ZaberStatus.ComponentStatus.iLastCommand.P_CommandStatus.LastCommandMessage := Base.F_GetLastWordInString(__POUNAME());
END_IF

IF NOT _DispatchValid() THEN
	RETURN;
ELSE
	_BuildCommandStringNoArgs();
	
	IF iBufferSend <> 0 AND __QUERYINTERFACE(iBufferSend, testIBufferSend) THEN
		iBufferSend.AddObject(RefObject := ZaberCommand);
	END_IF
END_IF
END_METHOD

METHOD io_info
IF ZaberStatus.ComponentStatus.iLastCommand <> 0 THEN
	ZaberStatus.ComponentStatus.iLastCommand.P_CommandStatus.LastCommandMessage := Base.F_GetLastWordInString(__POUNAME());
END_IF

IF NOT _DispatchValid() THEN
	RETURN;
ELSE
	_BuildCommandStringNoArgs();
	
	IF iBufferSend <> 0 AND __QUERYINTERFACE(iBufferSend, testIBufferSend) THEN
		iBufferSend.AddObject(RefObject := ZaberCommand);
	END_IF
END_IF
END_METHOD

METHOD lockstep_get
VAR_INPUT
	LockstepGroup	: USINT := 1; // The address of the lockstep group must be in the range 1 to lockstep.numgroups; lockstep.numgroups: the number of lockstep groupss; Valid Values: 0 to 2
//	Axis			: USINT := 1; //        The secondary axis to get the setting value for (optional).  The first secondary axis is labelled "b", the second "c", and so on
	Setting			: STRING(GPL_Zaber.STRING_LENGTH) := 'twist'; // Must be one of offset, parking.state, tolerance, or twist
END_VAR
IF ZaberStatus.ComponentStatus.iLastCommand <> 0 THEN
	ZaberStatus.ComponentStatus.iLastCommand.P_CommandStatus.LastCommandMessage := Base.F_GetLastWordInString(__POUNAME());
END_IF

IF NOT _DispatchValid() THEN
	RETURN;
ELSE
	_ClearTempString();
	ZaberCommand.stringval := Tc2_Standard.CONCAT(STR1 := ZaberConfiguration.sControllerRef, STR2 := ' ');
	ZaberCommand.stringval := Tc2_Standard.CONCAT(STR1 := ZaberCommand.stringval, STR2 := Base.F_GetFirstWordInString(sInput := SUPER^._iCommandConfiguration[ZaberStatus.ZaberMethodDispatch].P_CommandConfiguration.CommandDescription));
	ZaberCommand.stringval := Tc2_Standard.CONCAT(STR1 := ZaberCommand.stringval, STR2 := ' ');
	ZaberCommand.stringval := Tc2_Standard.CONCAT(STR1 := ZaberCommand.stringval, STR2 := USINT_TO_STRING(LockstepGroup));
	ZaberCommand.stringval := Tc2_Standard.CONCAT(STR1 := ZaberCommand.stringval, STR2 := ' ');
	ZaberCommand.stringval := Tc2_Standard.CONCAT(STR1 := ZaberCommand.stringval, STR2 := F_GetAllButFirstWord(sInput := SUPER^._iCommandConfiguration[ZaberStatus.ZaberMethodDispatch].P_CommandConfiguration.CommandDescription));
 	ZaberCommand.stringval := Tc2_Standard.CONCAT(STR1 := ZaberCommand.stringval, STR2 := ' ');
// 	ZaberCommand.stringval := Tc2_Standard.CONCAT(STR1 := ZaberCommand.stringval, STR2 := USINT_TO_STRING(Axis));
//	ZaberCommand.stringval := Tc2_Standard.CONCAT(STR1 := ZaberCommand.stringval, STR2 := ' ');
	ZaberCommand.stringval := Tc2_Standard.CONCAT(STR1 := ZaberCommand.stringval, STR2 := Setting);
	
	IF iBufferSend <> 0 AND __QUERYINTERFACE(iBufferSend, testIBufferSend) THEN
		iBufferSend.AddObject(RefObject := ZaberCommand);
	END_IF
END_IF
END_METHOD

METHOD lockstep_home
VAR_INPUT
	LockstepGroup	: USINT := 1; // The address of the lockstep group must be in the range 1 to lockstep.numgroups; lockstep.numgroups: the number of lockstep groupss; Valid Values: 0 to 2
END_VAR
IF ZaberStatus.ComponentStatus.iLastCommand <> 0 THEN
	ZaberStatus.ComponentStatus.iLastCommand.P_CommandStatus.LastCommandMessage := Base.F_GetLastWordInString(__POUNAME());
END_IF

IF NOT _DispatchValid() THEN
	RETURN;
ELSE
	_ClearTempString();
	ZaberCommand.stringval := Tc2_Standard.CONCAT(STR1 := ZaberConfiguration.sControllerRef, STR2 := ' ');
	ZaberCommand.stringval := Tc2_Standard.CONCAT(STR1 := ZaberCommand.stringval, STR2 := Base.F_GetFirstWordInString(sInput := SUPER^._iCommandConfiguration[ZaberStatus.ZaberMethodDispatch].P_CommandConfiguration.CommandDescription));
	ZaberCommand.stringval := Tc2_Standard.CONCAT(STR1 := ZaberCommand.stringval, STR2 := ' ');
	ZaberCommand.stringval := Tc2_Standard.CONCAT(STR1 := ZaberCommand.stringval, STR2 := USINT_TO_STRING(LockstepGroup));
	ZaberCommand.stringval := Tc2_Standard.CONCAT(STR1 := ZaberCommand.stringval, STR2 := ' ');
	ZaberCommand.stringval := Tc2_Standard.CONCAT(STR1 := ZaberCommand.stringval, STR2 := F_GetAllButFirstWord(sInput := SUPER^._iCommandConfiguration[ZaberStatus.ZaberMethodDispatch].P_CommandConfiguration.CommandDescription));
	
	IF iBufferSend <> 0 AND __QUERYINTERFACE(iBufferSend, testIBufferSend) THEN
		iBufferSend.AddObject(RefObject := ZaberCommand);
	END_IF
END_IF
END_METHOD

